METHOD metDI_RevisionSwitchOk
VAR_INPUT
    ITF_IN		:	CtaSysIO.ITF_IO;
END_VAR
VAR	
	ITF_DI		:	CtaSysIO.ITF_DI;
END_VAR
IF ITF_IN <> 0 THEN
	ITF_RevisionSwitchOk := ITF_IN;
	IF __QUERYINTERFACE(ITF_RevisionSwitchOk,ITF_DI) THEN
		xInActuatorRevisionSwitchOn := ITF_DI.proValue;
	END_IF
ELSE
	xInActuatorRevisionSwitchOn := 0;
END_IF
END_METHOD

PROPERTY proNotShowDI_RevisionSwitchOk : BOOL
GET
proNotShowDI_RevisionSwitchOk := NOT scParameter.scInSAtRevisionSwitch.fbxEnable.xValue OR scParameter.scInSAtRevisionSwitch.fbxInputMb.xValue;
END_GET
END_PROPERTY

PROPERTY proGetDI_RevisionSwitchOK : BOOL
GET
proGetDI_RevisionSwitchOK := xInActuatorRevisionSwitchOn;
END_GET
END_PROPERTY

PROPERTY proRevisionSwitch_ITF : CtaSysIO.ITF_IO
GET
proRevisionSwitch_ITF := ITF_RevisionSwitchOk;
END_GET
END_PROPERTY

PROPERTY proGetDI_FuseOK : BOOL
GET
proGetDI_FuseOK := xInFuseOk;
END_GET
END_PROPERTY

METHOD metDI_FuseOK
VAR_INPUT
    ITF_IN		:	CtaSysIO.ITF_IO;
END_VAR
VAR	
	ITF_DI		:	CtaSysIO.ITF_DI;
END_VAR
IF ITF_IN <> 0 THEN
	ITF_FuseOk := ITF_IN;
	IF __QUERYINTERFACE(ITF_FuseOk,ITF_DI) THEN
		xInFuseOk := ITF_DI.proValue;
	END_IF
ELSE
	xInFuseOk := 0;	
END_IF
END_METHOD

PROPERTY proNotShowDI_FuseOk : BOOL
GET
proNotShowDI_FuseOk := NOT scParameter.scFuse.fbxEnable.xValue OR scParameter.scFuse.fbxInputMb.xValue;
END_GET
END_PROPERTY

PROPERTY proFuse_ITF : CtaSysIO.ITF_IO
GET
proFuse_ITF := ITF_FuseOk;
END_GET
END_PROPERTY

METHOD metDI_ActuatorHand
VAR_INPUT
    ITF_IN		:	CtaSysIO.ITF_IO;
END_VAR
VAR	
	ITF_DI		:	CtaSysIO.ITF_DI;
END_VAR
IF ITF_IN <> 0 THEN
	ITF_ActuatorHand := ITF_IN;
	IF __QUERYINTERFACE(ITF_ActuatorHand,ITF_DI) THEN
		xInActuatorHand := ITF_DI.proValue;
	END_IF
ELSE	
	xInActuatorHand := 0;
END_IF
END_METHOD

PROPERTY proNotShowDI_ActuatorHand : BOOL
GET
proNotShowDI_ActuatorHand := NOT scParameter.scInSAtHand.fbxEnable.xValue OR scParameter.scInSAtHand.fbxInputMb.xValue;
END_GET
END_PROPERTY

PROPERTY proGetDI_ActuatorHand : BOOL
GET
proGetDI_ActuatorHand := xInActuatorHand;
END_GET
END_PROPERTY

PROPERTY proHandModul_ITF : CtaSysIO.ITF_IO
GET
proHandModul_ITF := ITF_ActuatorHand;
END_GET
END_PROPERTY

METHOD metDI_IsReady
VAR_INPUT
    ITF_IN		:	CtaSysIO.ITF_IO;
END_VAR
VAR	
	ITF_DI		:	CtaSysIO.ITF_DI;
END_VAR
IF ITF_IN <> 0 THEN
	ITF_ActuatorIsReady := ITF_IN;
	IF __QUERYINTERFACE(ITF_ActuatorIsReady,ITF_DI) THEN
		xInActuatorIsReady := ITF_DI.proValue;
	END_IF
ELSE
	xInActuatorIsReady := 0;
END_IF
END_METHOD

PROPERTY proNotShowDI_Ready : BOOL
GET
proNotShowDI_Ready := NOT scParameter.scInSAtReady.fbxEnable.xValue OR scParameter.scInSAtReady.fbxInputMb.xValue;
END_GET
END_PROPERTY

PROPERTY proGetDI_IsReady : BOOL
GET
proGetDI_IsReady := xInActuatorIsReady;
END_GET
END_PROPERTY

PROPERTY proActuatorReady_ITF : CtaSysIO.ITF_IO
GET
proActuatorReady_ITF := ITF_ActuatorIsReady;
END_GET
END_PROPERTY

PROPERTY proActuatorFuse_ITF : CtaSysIO.ITF_IO
GET
proActuatorFuse_ITF := ITF_ActuatorFuseOk;
END_GET
END_PROPERTY

METHOD metDI_ActuatorFuseOk
VAR_INPUT
    ITF_IN		:	CtaSysIO.ITF_IO;
END_VAR
VAR	
	ITF_DI		:	CtaSysIO.ITF_DI;
END_VAR
IF ITF_IN <> 0 THEN
	ITF_ActuatorFuseOk := ITF_IN;
	IF __QUERYINTERFACE(ITF_ActuatorFuseOk,ITF_DI) THEN
		xInActuatorFuseOk := ITF_DI.proValue;
	END_IF
ELSE	
	xInActuatorFuseOk := 0;
END_IF
END_METHOD

PROPERTY proNotShowDI_ActuatorFuseOk : BOOL
GET
proNotShowDI_ActuatorFuseOk := NOT scParameter.scActuatorFuse.fbxEnable.xValue OR scParameter.scActuatorFuse.fbxInputMb.xValue;
END_GET
END_PROPERTY

PROPERTY proGetDI_ActuatorFuseOk : BOOL
GET
proGetDI_ActuatorFuseOk := xInActuatorFuseOk;
END_GET
END_PROPERTY

METHOD metAI_ActualPosition
VAR_INPUT
    ITF_IN		:	CtaSysIO.ITF_IO;
END_VAR
VAR	
	ITF_AI		:	CtaSysIO.ITF_AI;
END_VAR
IF ITF_IN <> 0 THEN
	ITF_ActualPosition := ITF_IN;
	IF __QUERYINTERFACE(ITF_ActualPosition,ITF_AI) THEN
		rInActualPosition := ITF_AI.proValue;
	END_IF
ELSE	
	rInActualPosition := 0;
END_IF
END_METHOD

PROPERTY proNotShowAI_ActualPosition : BOOL
GET
proNotShowAI_ActualPosition := NOT scParameter.scInSAtActualPosition.fbxEnable.xValue OR scParameter.scInSAtActualPosition.fbxInputMb.xValue;
END_GET
END_PROPERTY

PROPERTY proGetAI_ActualPosition : REAL
GET
proGetAI_ActualPosition := rInActualPosition;
END_GET
END_PROPERTY

PROPERTY proActualPosition_ITF : CtaSysIO.ITF_IO
GET
proActualPosition_ITF := ITF_ActualPosition;
END_GET
END_PROPERTY

PROPERTY proOnY_ITF : CtaSysIO.ITF_IO
GET
proOnY_ITF := ITF_rOnY;
END_GET
END_PROPERTY

METHOD metAO_OnY : REAL
VAR_INPUT
    ITF_IN		:	CtaSysIO.ITF_IO;
END_VAR
VAR	
	ITF_AO		:	CtaSysIO.ITF_AO;
END_VAR
IF ITF_IN <> 0 THEN
	ITF_rOnY := ITF_IN;	
	IF __QUERYINTERFACE(ITF_rOnY,ITF_AO) THEN		
		ITF_AO.proValue := rOnY;
	END_IF	
ELSE
	metAO_OnY := rOnY;
END_IF
END_METHOD

METHOD metDO_xOnAuf : BOOL
VAR_INPUT
    ITF_IN		:	CtaSysIO.ITF_IO;
END_VAR
VAR	
	ITF_DO		:	CtaSysIO.ITF_DO;
END_VAR
IF ITF_IN <> 0 THEN	
	ITF_xOnAuf := ITF_IN;
	IF __QUERYINTERFACE(ITF_xOnAuf,ITF_DO) THEN		
		ITF_DO.proValue := xOnAuf;
	END_IF	
ELSE
	metDO_xOnAuf := xOnAuf;
END_IF
END_METHOD

PROPERTY proOnOpen_ITF : CtaSysIO.ITF_IO
GET
proOnOpen_ITF := ITF_xOnAuf;
END_GET
END_PROPERTY

PROPERTY proOnClose_ITF : CtaSysIO.ITF_IO
GET
proOnClose_ITF := ITF_xOnZu;
END_GET
END_PROPERTY

METHOD metDO_xOnZu : BOOL
VAR_INPUT
    ITF_IN		:	CtaSysIO.ITF_IO;
END_VAR
VAR	
	ITF_DO		:	CtaSysIO.ITF_DO;
END_VAR
IF ITF_IN <> 0 THEN	
	ITF_xOnZu := ITF_IN;
	IF __QUERYINTERFACE(ITF_xOnZu,ITF_DO) THEN		
		ITF_DO.proValue := xOnZu;
	END_IF	
ELSE
	metDO_xOnZu := xOnZu;
END_IF
END_METHOD

PROPERTY proOnY : REAL
GET
proOnY := rOnY;
END_GET
END_PROPERTY

ACTION actPrioOfControll:
(* get Controll request *)
xReleaseControllPrio := SEL(xRelease,xReleaseFromModBus,xRelease);  // xRelease request from Software has prio
rReleaseControllPrio := SEL(xRelease,rReleaseFromModBus,rRelease);  // rRelease request from Software has prio

(* Get state from Input or ModBus *)

(* Actuall Position from AI *)
// Value Actual Position 0 if not Enabled
rActualPosition						:= SEL(scParameter.scInSAtActualPosition.fbxEnable.xValue	,rOnY	,SEL(scParameter.scInSAtActualPosition.fbxInputMb.xValue	,rInActualPosition				,rInActualPositionMb			)); 
(* Actuator is Open *)
// Flag RückIsOpen False if not Enabled
xRückIsOpen							:= SEL(scParameter.scInSAtRükOpen.fbxEnable.xValue			,FALSE	,SEL(scParameter.scInSAtRükOpen.fbxInputMb.xValue			,xInRükIsOpen					,xInRükIsOpenMb					));
(* Actuator is Closed *)
// Flag RückIsClosed False if not Enabled
xRückIsClosed						:= SEL(scParameter.scInSAtRükClosed.fbxEnable.xValue		,FALSE	,SEL(scParameter.scInSAtRükClosed.fbxInputMb.xValue			,xInRükIsClosed					,xInRükIsClosedMb				));
(* Fuse ok *)
// Flag FuseOk True if not Enabled
xFuseOk								:= SEL(scParameter.scFuse.fbxEnable.xValue					,TRUE	,SEL(scParameter.scFuse.fbxInputMb.xValue					,xInFuseOk						,xInFuseOkMb                	));                     
(* Motor fuse ok *)
// Flag MotorFuseOk True if not Enabled
xActuatorFuseOk						:= SEL(scParameter.scActuatorFuse.fbxEnable.xValue			,TRUE	,SEL(scParameter.scActuatorFuse.fbxInputMb.xValue			,xInActuatorFuseOk				,xInActuatorFuseOkMb           	));
(* Motor is ready *)
// Flag MotorIsReady True if not Enabled
xActuatorIsReady					:= SEL(scParameter.scInSAtReady.fbxEnable.xValue			,TRUE	,SEL(scParameter.scInSAtReady.fbxInputMb.xValue				,xInActuatorIsReady				,xInActuatorIsReadyMb          	)); 
(* Revision Switch *)
// Flag MotorRevisionSwitchOn True if not Enabled
xActuatorRevisionSwitchOn			:= SEL(scParameter.scInSAtRevisionSwitch.fbxEnable.xValue	,TRUE	,SEL(scParameter.scInSAtRevisionSwitch.fbxInputMb.xValue	,xInActuatorRevisionSwitchOn	,xInActuatorRevisionSwitchOnMb 	));
xActuatorRevisionSwitchOff			:= NOT xActuatorRevisionSwitchOn;
(* Motor is hand *)
// Flag MotorHand False if not Enabled
xActuatorHand						:= SEL(scParameter.scInSAtHand.fbxEnable.xValue				,FALSE	,SEL(scParameter.scInSAtHand.fbxInputMb.xValue				,xInActuatorHand				,xInActuatorHandMb             	));
END_ACTION

ACTION actResetOnDisable:
TP_StartOeffnungVorlauf.PT  := T#0MS;
TP_StartOeffnungVorlauf.IN  := FALSE ;  
TP_StartOeffnungVorlauf();
                          
TP_Open.PT					:= T#0S;
TP_Open.IN					:= FALSE;
TP_Open();                  
TP_Close.PT					:= T#0S;  
TP_Close.IN					:= FALSE;
TP_Open();                  
                            
rActualPosition				:= 0	;
xRückIsOpen					:= FALSE;
xRückIsClosed				:= FALSE;
xFuseOk						:= FALSE;    
xActuatorFuseOk				:= FALSE;
xActuatorIsReady			:= FALSE;
xActuatorRevisionSwitchOn	:= FALSE;
xActuatorHand				:= FALSE;
END_ACTION

PROPERTY proOnAuf : BOOL
GET
proOnAuf := xOnAuf;
END_GET
END_PROPERTY

PROPERTY proOnZu : BOOL
GET
proOnZu := xOnZu;
END_GET
END_PROPERTY

//FB_Init ist immer implizit verfügbar und wird primär für die Initialisierung verwendet.
//Der Rückgabewert wird nicht ausgewertet. Für gezielte Einflussnahme können Sie
//die Methoden explizit deklarieren und darin mit dem Standard-Initialisierungscode 
//zusätzlichen Code bereitstellen. Sie können den Rückgabewert auswerten.
METHOD FB_INIT: BOOL
VAR_INPUT    
bInitRetains: BOOL; // TRUE: Die Retain-Variablen werden initialisiert (Reset warm / Reset kalt)    
bInCopyCode: BOOL;  // TRUE: Die Instanz wird danach in den Kopiercode kopiert (Online-Change)
END_VAR
VAR
    ITF_AT_THIS             :   ITF_STELLANTRIEB;
    ITF_AT_QUERRY           :   ITF_STELLANTRIEB;
END_VAR
IF NOT bInCopyCode THEN
    ITF_AT_THIS := THIS^;
    IF __QUERYINTERFACE(ITF_AT_THIS,ITF_AT_QUERRY) THEN
        diArrayPosition := GVL_StellAntrieb.fbStellAntrieb_Collector.metRegistry(ITF_AT_QUERRY);
    END_IF;
END_IF;
END_METHOD

PROPERTY proEn : BOOL
SET
xIsEnabled := proEn;
END_SET
GET
proEn := xIsEnabled;
END_GET
END_PROPERTY

PROPERTY proEnSymbol : STRING
GET
IF xIsEnabled THEN
    proEnSymbol := 'CtaVisSymbols.ImagePool.CheckboxChecked_blue';
ELSE    
    proEnSymbol := 'CtaVisSymbols.ImagePool.CheckboxUnchecked_withe'; 
END_IF;
END_GET
END_PROPERTY

ACTION actTrendLog:
(* Stellwert Digital zu *)		
fbTrendxOnZu.ENABLE 			:=	scParameter.scBase.fbxEnable.proValue AND
									scParameter.scInfluxDb.fbxEnable.proValue;
fbTrendxOnZu.KEY   				:= 	CONCAT(stObjID,'_xOnZu');
fbTrendxOnZu.SET_VALUE			:=	xOnZu;

(* Rückmeldung Digital zu *)
fbTrendxRückClosed.ENABLE 		:=	scParameter.scBase.fbxEnable.proValue AND
									scParameter.scInfluxDb.fbxEnable.proValue;
fbTrendxRückClosed.KEY   		:= 	CONCAT(stObjID,'_xRückIsClosed');
fbTrendxRückClosed.SET_VALUE	:=	xRückIsClosed;

(* Stellwert Digital auf *)
fbTrendxOnAuf.ENABLE 			:=	scParameter.scBase.fbxEnable.proValue AND
									scParameter.scInfluxDb.fbxEnable.proValue;
fbTrendxOnAuf.KEY   			:= 	CONCAT(stObjID,'_xOnAuf');
fbTrendxOnAuf.SET_VALUE			:=	xOnAuf;

(* Rückmeldung Digital auf *)
fbTrendxRückIsOpen.ENABLE 		:=	scParameter.scBase.fbxEnable.proValue AND
									scParameter.scInfluxDb.fbxEnable.proValue;
fbTrendxRückIsOpen.KEY   		:= 	CONCAT(stObjID,'_xRückIsOpen');
fbTrendxRückIsOpen.SET_VALUE	:=	xRückIsOpen;

(* Stellwert Analog *)
fbTrendrOnY.ENABLE 				:=	scParameter.scBase.fbxEnable.proValue AND
									scParameter.scInfluxDb.fbxEnable.proValue;
fbTrendrOnY.KEY   				:= 	CONCAT(stObjID,'_rOnY');
fbTrendrOnY.SET_VALUE			:=	rOnY;

(* Istwert Analog *)
fbTrendrIsOnY.ENABLE 			:=	scParameter.scBase.fbxEnable.proValue AND
									scParameter.scInfluxDb.fbxEnable.proValue;
fbTrendrIsOnY.KEY   			:= 	CONCAT(stObjID,'_rIsOnY');
fbTrendrIsOnY.SET_VALUE			:=	proIsOnY;

(* Fehler *)
fbTrendxError.ENABLE 			:=	scParameter.scBase.fbxEnable.proValue AND
									scParameter.scInfluxDb.fbxEnable.proValue;
fbTrendxError.KEY   			:= 	CONCAT(stObjID,'_xError');
fbTrendxError.SET_VALUE			:=	xIsError;
END_ACTION

ACTION actReport:
(* EWI Manager *)
fbReportManager(	stErrorInitReportTextListIn		:=	ADR(GlobalKonstant.stReportTextListError),
					stWarningInitReportTextListIn	:=	ADR(GlobalKonstant.stReportTextListWarning),
					stInfoInitReportTextListIn		:=	ADR(GlobalKonstant.stReportTextListInfo),
					scReportNr						:=	scEWI);
(* Errors *)                        
		(* Stellwert Rückmeldung *)
		ayErrorReporter[1].proPrio  := 3;
		ayErrorReporter[1].metReport(     		xSetReportIn					:= xErrorDiffAI AND scParameter.scInSAtActualPosition.fbxDoesAlarm.proValue AND scParameter.scInSAtActualPosition.fbxEnable.proValue,
												iReportID						:= 1,
												enReportTypeIn					:= CtaAppReport.enReportType.Error,  
												enReportAcknowledgeTypeIn   	:= scParameter.scInSAtActualPosition.fbiTypeOfAck.proValue,
												tDelay							:= T#0S, 
												ITF_BMK_IN						:= THIS^,			              
												pstReportTextListIn				:= ADR(GlobalKonstant.stReportTextListError),
												stOptionalReportText		    := '',   
												iRetryTilReportLock 		    := scParameter.scInSAtActualPosition.fbiMaxErrorRetryAllowed.proValue, 
												xResetCount         		    := FALSE,  
												tReset						    := T#24H); 		

		(* Stellventil keine rückmeldung Zu *) 
		ayErrorReporter[2].proPrio  := 3;   
        ayErrorReporter[2].metReport(     		xSetReportIn					:= xErrorCloseDI AND scParameter.scInSAtRükClosed.fbxDoesAlarm.proValue AND scParameter.scInSAtRükClosed.fbxEnable.proValue,
												iReportID						:= 2,
												enReportTypeIn					:= CtaAppReport.enReportType.Error,  
												enReportAcknowledgeTypeIn   	:= scParameter.scInSAtRükClosed.fbiTypeOfAck.proValue,
												tDelay							:= T#0S, 
												ITF_BMK_IN						:= THIS^,			              
												pstReportTextListIn				:= ADR(GlobalKonstant.stReportTextListError),
												stOptionalReportText		    := '',   
												iRetryTilReportLock 		    := scParameter.scInSAtRükClosed.fbiMaxErrorRetryAllowed.proValue, 
												xResetCount         		    := FALSE,  
												tReset						    := T#24H); 	  
		(* Stellventil keine rückmeldung Auf *)
		ayErrorReporter[3].proPrio  := 3; 
		ayErrorReporter[3].metReport(     		xSetReportIn					:= xErrorOpenDI AND scParameter.scInSAtRükOpen.fbxDoesAlarm.proValue AND scParameter.scInSAtRükOpen.fbxEnable.proValue,
												iReportID						:= 3,
												enReportTypeIn					:= CtaAppReport.enReportType.Error,  
												enReportAcknowledgeTypeIn   	:= scParameter.scInSAtRükOpen.fbiTypeOfAck.proValue,
												tDelay							:= T#1S, 
												ITF_BMK_IN						:= THIS^,			              
												pstReportTextListIn				:= ADR(GlobalKonstant.stReportTextListError),
												stOptionalReportText		    := '',   
												iRetryTilReportLock 		    := scParameter.scInSAtRükOpen.fbiMaxErrorRetryAllowed.proValue, 
												xResetCount         		    := FALSE,  
												tReset						    := T#24H);
		(* Monitoring digitaler Stellwert *)
		ayErrorReporter[4].proPrio  := 3;    
		ayErrorReporter[4].metReport(     		xSetReportIn					:= xErrorDiRük AND scParameter.scBase.fbxEnDigitalMonitoring.proValue,
												iReportID						:= 4,
												enReportTypeIn					:= CtaAppReport.enReportType.Error,  
												enReportAcknowledgeTypeIn   	:= CtaAppReport.enReportacknowledgeType.Auto,
												tDelay							:= T#1S, 
												ITF_BMK_IN						:= THIS^,			              
												pstReportTextListIn				:= ADR(GlobalKonstant.stReportTextListError),
												stOptionalReportText		    := '',   
												iRetryTilReportLock 		    := 0, 
												xResetCount         		    := FALSE,  
												tReset						    := T#24H);
		(* Monitoring analoger Stellwert *)
		ayErrorReporter[5].proPrio  := 3;     
		ayErrorReporter[5].metReport(     		xSetReportIn					:= xErrorAIRük AND scParameter.scBase.fbxEnAnalogMonitoring.proValue,
												iReportID						:= 5,
												enReportTypeIn					:= CtaAppReport.enReportType.Error,  
												enReportAcknowledgeTypeIn   	:= CtaAppReport.enReportacknowledgeType.Auto,
												tDelay							:= T#1S, 
												ITF_BMK_IN						:= THIS^,			              
												pstReportTextListIn				:= ADR(GlobalKonstant.stReportTextListError),
												stOptionalReportText		    := '',   
												iRetryTilReportLock 		    := 0, 
												xResetCount         		    := FALSE,  
												tReset						    := T#24H);                    
		(* Error Fuse *)
		ayErrorReporter[6].proPrio  := 2;    
		ayErrorReporter[6].metReport(     		xSetReportIn					:= NOT xFuseOk AND scParameter.scFuse.fbxDoesAlarm.proValue AND scParameter.scFuse.fbxEnable.proValue,
												iReportID						:= 6,
												enReportTypeIn					:= CtaAppReport.enReportType.Error,  
												enReportAcknowledgeTypeIn   	:= CtaAppReport.enReportacknowledgeType.Auto,
												tDelay							:= T#1S, 
												ITF_BMK_IN						:= THIS^,			              
												pstReportTextListIn				:= ADR(GlobalKonstant.stReportTextListError),
												stOptionalReportText		    := '',   
												iRetryTilReportLock 		    := 0, 
												xResetCount         		    := FALSE,  
												tReset						    := T#24H);
                                                
		(* Error Actuator Fuse *)
		ayErrorReporter[7].proPrio  := 2;    
		ayErrorReporter[7].metReport(     		xSetReportIn					:= NOT xActuatorFuseOk AND scParameter.scActuatorFuse.fbxDoesAlarm.proValue AND scParameter.scActuatorFuse.fbxEnable.proValue,
												iReportID						:= 7,
												enReportTypeIn					:= CtaAppReport.enReportType.Error,  
												enReportAcknowledgeTypeIn   	:= CtaAppReport.enReportacknowledgeType.Auto,
												tDelay							:= T#1S, 
												ITF_BMK_IN						:= THIS^,			              
												pstReportTextListIn				:= ADR(GlobalKonstant.stReportTextListError),
												stOptionalReportText		    := '',   
												iRetryTilReportLock 		    := 0, 
												xResetCount         		    := FALSE,  
												tReset						    := T#24H);                                                

		(* Config Error *)
		ayErrorReporter[8].proPrio  := 1;    
		ayErrorReporter[8].metReport(     		xSetReportIn					:= xConfigError,
												iReportID						:= 8,
												enReportTypeIn					:= CtaAppReport.enReportType.Error,  
												enReportAcknowledgeTypeIn   	:= CtaAppReport.enReportacknowledgeType.Quit,
												tDelay							:= T#1S, 
												ITF_BMK_IN						:= THIS^,			              
												pstReportTextListIn				:= ADR(GlobalKonstant.stReportTextListError),
												stOptionalReportText		    := '',   
												iRetryTilReportLock 		    := 0, 
												xResetCount         		    := FALSE,  
												tReset						    := T#24H);                                           
(* Warnungen *)
		(* Warnung Revisionsschalter Aus *)
		ayWarningReporter[1].proPrio  := 1;
		ayWarningReporter[1].proHandLokal :=   	xActuatorRevisionSwitchOff; 
		ayWarningReporter[1].metReport(			xSetReportIn					:= xActuatorRevisionSwitchOff,
												iReportID						:= 1,
												enReportTypeIn					:= CtaAppReport.enReportType.Warning,  
												enReportAcknowledgeTypeIn   	:= CtaAppReport.enReportAcknowledgeType.Auto,
												tDelay							:= T#0S, 
												ITF_BMK_IN						:= THIS^,			              
												pstReportTextListIn				:= ADR(GlobalKonstant.stReportTextListWarning),
												stOptionalReportText		    := '',   
												iRetryTilReportLock 		    := 0, 
												xResetCount         		    := FALSE,  
												tReset						    := T#0S);     

		(* Warnung Hand Aus *)
		ayWarningReporter[2].proPrio  := 3;        
		ayWarningReporter[2].proHandLokal :=    xIsHandOff; 
		ayWarningReporter[2].metReport(			xSetReportIn					:= xIsHandOff,
												iReportID						:= 2,
												enReportTypeIn					:= CtaAppReport.enReportType.Warning,  
												enReportAcknowledgeTypeIn   	:= CtaAppReport.enReportAcknowledgeType.Auto,
												tDelay							:= T#0S, 
												ITF_BMK_IN						:= THIS^,			              
												pstReportTextListIn				:= ADR(GlobalKonstant.stReportTextListWarning),
												stOptionalReportText		    := '',   
												iRetryTilReportLock 		    := 0, 
												xResetCount         		    := FALSE,  
												tReset						    := T#0S);                                  
                                
        (* Warnung Hand Ein *)
		ayWarningReporter[3].proPrio  := 3;    
		ayWarningReporter[3].proHandLokal :=    xIsHandOn;
		ayWarningReporter[3].metReport(			xSetReportIn					:= xIsHandOn,
												iReportID						:= 3,
												enReportTypeIn					:= CtaAppReport.enReportType.Warning,  
												enReportAcknowledgeTypeIn   	:= CtaAppReport.enReportAcknowledgeType.Auto,
												tDelay							:= T#0S, 
												ITF_BMK_IN						:= THIS^,			              
												pstReportTextListIn				:= ADR(GlobalKonstant.stReportTextListWarning),
												stOptionalReportText		    := '',   
												iRetryTilReportLock 		    := 0, 
												xResetCount         		    := FALSE,  
												tReset						    := T#0S);   
 
        (* Warnung Handmodul Actuator *)
		ayWarningReporter[4].proPrio  := 4;    
		ayWarningReporter[4].proHandLokal :=    xActuatorHand;
		ayWarningReporter[4].metReport(			xSetReportIn					:= xActuatorHand,
												iReportID						:= 4,
												enReportTypeIn					:= CtaAppReport.enReportType.Warning,  
												enReportAcknowledgeTypeIn   	:= CtaAppReport.enReportAcknowledgeType.Auto,
												tDelay							:= T#0S, 
												ITF_BMK_IN						:= THIS^,			              
												pstReportTextListIn				:= ADR(GlobalKonstant.stReportTextListWarning),
												stOptionalReportText		    := '',   
												iRetryTilReportLock 		    := 0, 
												xResetCount         		    := FALSE,  
												tReset						    := T#0S);                                                   
(* Sync Reports *)                                         
FOR difor := LOWER_BOUND(ayErrorReporter,1) TO UPPER_BOUND(ayErrorReporter,1) DO
	fbReportManager.metSyncReporter(ayErrorReporter[difor]);	
END_FOR;
FOR difor := LOWER_BOUND(ayWarningReporter,1) TO UPPER_BOUND(ayWarningReporter,1) DO
	fbReportManager.metSyncReporter(ayWarningReporter[difor]);	
END_FOR;
                                                                             
_xIsError   := scEWI.iError <> 0;
_xIsWarning := scEWI.iWarning <> 0;
END_ACTION

{attribute 'monitoring' := 'variable'}
PROPERTY proAcknowlege : BOOL
GET
proAcknowlege := NOT proIsError;
END_GET
END_PROPERTY

{attribute 'monitoring' := 'variable'}
PROPERTY proAvailable : BOOL
GET
proAvailable := proIsReady;
END_GET
END_PROPERTY

{attribute 'monitoring' := 'variable'}
PROPERTY proLockDown : BOOL
GET
proLockDown := proIsError;
END_GET
END_PROPERTY

END_FUNCTION_BLOCK

// 30 Program Organization Units/Abstracte Bausteine/fbAntriebTabellenInfo
{attribute 'hide'} 
FUNCTION_BLOCK INTERNAL ABSTRACT fbAntriebTabellenInfo EXTENDS CtaAppBmk.fbBMK IMPLEMENTS ITF_STELLANTRIEB_TABELLE_INFO

PROPERTY proOnAuf : BOOL
GET
END_GET
END_PROPERTY

PROPERTY proStateSymbol : STRING
GET
END_GET
END_PROPERTY

PROPERTY proEnSymbol : STRING
GET
END_GET
END_PROPERTY

PROPERTY proIsOn : BOOL
GET
END_GET
END_PROPERTY

PROPERTY proIsOnY : REAL
GET
END_GET
END_PROPERTY

PROPERTY proOn : BOOL
GET
END_GET
END_PROPERTY

PROPERTY proOnY : REAL
GET
END_GET
END_PROPERTY

PROPERTY proOnZu : BOOL
GET
END_GET
END_PROPERTY

PROPERTY proRükIsClosed : BOOL
GET
END_GET
END_PROPERTY

PROPERTY proRükIsOpen : BOOL
GET
END_GET
END_PROPERTY

END_FUNCTION_BLOCK

// 21 Interface/ITF_STELLANTRIEB_TABELLE_INFO
INTERFACE INTERNAL ITF_STELLANTRIEB_TABELLE_INFO EXTENDS CtaAppBmk.ITF_BMK

PROPERTY proRükIsOpen : BOOL
GET
END_GET
END_PROPERTY

PROPERTY proRükIsClosed : BOOL
GET
END_GET
END_PROPERTY

PROPERTY INTERNAL proStateSymbol : STRING
GET
END_GET
END_PROPERTY

PROPERTY INTERNAL proEnSymbol : STRING
GET
END_GET
END_PROPERTY

PROPERTY proOnZu : BOOL
GET
END_GET
END_PROPERTY

PROPERTY proIsOnY : REAL
GET
END_GET
END_PROPERTY

PROPERTY proOnAuf : BOOL
GET
END_GET
END_PROPERTY

PROPERTY proOnY : REAL
GET
END_GET
END_PROPERTY

END_INTERFACE

// 21 Interface/ITF_STELLANTRIEB
INTERFACE ITF_STELLANTRIEB EXTENDS ITF_STELLANTRIEB_TABELLE_INFO,CtaAppModbusSpezifikation.ITF_MODBUS_SPEZIFIKATION

PROPERTY proAuto : BOOL
GET
END_GET
SET
END_SET
END_PROPERTY

PROPERTY proHandOff : BOOL
GET
END_GET
SET
END_SET
END_PROPERTY

PROPERTY proHandOn : BOOL
GET
END_GET
SET
END_SET
END_PROPERTY

PROPERTY proIsRegulatet : BOOL
GET
END_GET
END_PROPERTY

PROPERTY proIsError : BOOL
GET
END_GET
END_PROPERTY

PROPERTY proIsWarning : BOOL
GET
END_GET
END_PROPERTY

PROPERTY proIsEnabled : BOOL
GET
END_GET
END_PROPERTY

PROPERTY proIsHandOnOrOff : BOOL
GET
END_GET
END_PROPERTY

PROPERTY proIsReady : BOOL
GET
END_GET
END_PROPERTY

PROPERTY proHardWareHandModulAktive : BOOL
GET
END_GET
END_PROPERTY

PROPERTY proRevisionSwitchOk : BOOL
GET
END_GET
END_PROPERTY

PROPERTY proHandOnY : REAL
SET
END_SET
GET
END_GET
END_PROPERTY

PROPERTY proEn : BOOL
SET
END_SET
GET
END_GET
END_PROPERTY

PROPERTY proGetDI_RükIsOpen : BOOL
GET
END_GET
END_PROPERTY

PROPERTY proNotShowDI_RükIsOpen : BOOL
GET
END_GET
END_PROPERTY

PROPERTY proIsOpen_ITF : CtaSysIO.ITF_IO
GET
END_GET
END_PROPERTY

PROPERTY INTERNAL proGetDI_ActuatorHand : BOOL
GET
END_GET
END_PROPERTY

PROPERTY proNotShowDI_ActuatorHand : BOOL
GET
END_GET
END_PROPERTY

PROPERTY proHandModul_ITF : CtaSysIO.ITF_IO
GET
END_GET
END_PROPERTY

PROPERTY INTERNAL proGetDI_ActuatorFuseOk : BOOL
GET
END_GET
END_PROPERTY

PROPERTY proNotShowDI_ActuatorFuseOk : BOOL
GET
END_GET
END_PROPERTY

PROPERTY proActuatorFuse_ITF : CtaSysIO.ITF_IO
GET
END_GET
END_PROPERTY

PROPERTY INTERNAL proGetDI_IsReady : BOOL
GET
END_GET
END_PROPERTY

PROPERTY proNotShowDI_Ready : BOOL
GET
END_GET
END_PROPERTY

PROPERTY proActuatorReady_ITF : CtaSysIO.ITF_IO
GET
END_GET
END_PROPERTY

PROPERTY INTERNAL proGetDI_FuseOK : BOOL
GET
END_GET
END_PROPERTY

PROPERTY proNotShowDI_FuseOk : BOOL
GET
END_GET
END_PROPERTY

PROPERTY proFuse_ITF : CtaSysIO.ITF_IO
GET
END_GET
END_PROPERTY

PROPERTY INTERNAL proGetDI_RevisionSwitchOK : BOOL
GET
END_GET
END_PROPERTY

PROPERTY proNotShowDI_RevisionSwitchOk : BOOL
GET
END_GET
END_PROPERTY

PROPERTY proRevisionSwitch_ITF : CtaSysIO.ITF_IO
GET
END_GET
END_PROPERTY

PROPERTY proNotShowAI_ActualPosition : BOOL
GET
END_GET
END_PROPERTY

PROPERTY proGetAI_ActualPosition : REAL
GET
END_GET
END_PROPERTY

PROPERTY proActualPosition_ITF : CtaSysIO.ITF_IO
GET
END_GET
END_PROPERTY

PROPERTY proGetDI_RükIsClosed : BOOL
GET
END_GET
END_PROPERTY

PROPERTY proNotShowDI_RükIsClosed : BOOL
GET
END_GET
END_PROPERTY

PROPERTY proIsClosed_ITF : CtaSysIO.ITF_IO
GET
END_GET
END_PROPERTY

PROPERTY proOnOpen_ITF : CtaSysIO.ITF_IO
GET
END_GET
END_PROPERTY

PROPERTY proOnClose_ITF : CtaSysIO.ITF_IO
GET
END_GET
END_PROPERTY

PROPERTY proOnY_ITF : CtaSysIO.ITF_IO
GET
END_GET
END_PROPERTY

PROPERTY INTERNAL proAnzWarning : INT
GET
END_GET
END_PROPERTY

PROPERTY INTERNAL proITF_REPORTMANAGER : CtaAppReport.ITF_REPORTMANAGER
GET
END_GET
END_PROPERTY

PROPERTY INTERNAL proAnzInfo : INT
GET
END_GET
END_PROPERTY

PROPERTY INTERNAL proAnzError : INT
GET
END_GET
END_PROPERTY

PROPERTY INTERNAL proModbusTest : BOOL
SET
END_SET
GET
END_GET
END_PROPERTY

PROPERTY proModbusStateWord : REFERENCE TO ARRAY[0..3] OF WORD
GET
END_GET
END_PROPERTY

PROPERTY proModbusControllWord : REFERENCE TO ARRAY[0..3] OF WORD
GET
END_GET
END_PROPERTY

PROPERTY proConfigError : BOOL
GET
END_GET
END_PROPERTY

PROPERTY p_scActuatorFuse_fbxEnable : CtaSysConfig.ITF_DATATYPE;
GET
END_GET
END_PROPERTY

PROPERTY p_scActuatorFuse_fbxInputMb : CtaSysConfig.ITF_DATATYPE;
GET
END_GET
END_PROPERTY

PROPERTY p_scActuatorFuse_fbxDoesAlarm : CtaSysConfig.ITF_DATATYPE;
GET
END_GET
END_PROPERTY

PROPERTY p_scBase_fbxEnable : CtaSysConfig.ITF_DATATYPE;
GET
END_GET
END_PROPERTY

PROPERTY p_scBase_fbxControllMb : CtaSysConfig.ITF_DATATYPE;
GET
END_GET
END_PROPERTY

PROPERTY p_scBase_fbxInvertiert : CtaSysConfig.ITF_DATATYPE;
GET
END_GET
END_PROPERTY

PROPERTY p_scBase_fbxRegulatet : CtaSysConfig.ITF_DATATYPE;
GET
END_GET
END_PROPERTY

PROPERTY p_scBase_fbrYMin : CtaSysConfig.ITF_DATATYPE;
GET
END_GET
END_PROPERTY

PROPERTY p_scBase_fbrYMax : CtaSysConfig.ITF_DATATYPE;
GET
END_GET
END_PROPERTY

PROPERTY p_scBase_fbxEnStartPosition : CtaSysConfig.ITF_DATATYPE;
GET
END_GET
END_PROPERTY

PROPERTY p_scBase_fbrYStartPos : CtaSysConfig.ITF_DATATYPE;
GET
END_GET
END_PROPERTY

PROPERTY p_scBase_fbtStartPosTime : CtaSysConfig.ITF_DATATYPE;
GET
END_GET
END_PROPERTY

PROPERTY p_scBase_fbrYStopp : CtaSysConfig.ITF_DATATYPE;
GET
END_GET
END_PROPERTY

PROPERTY p_scBase_fbtYSettingTime : CtaSysConfig.ITF_DATATYPE;
GET
END_GET
END_PROPERTY

PROPERTY p_scBase_fbxEnDigitalValve : CtaSysConfig.ITF_DATATYPE;
GET
END_GET
END_PROPERTY

PROPERTY p_scBase_fbrHysteresisDigital : CtaSysConfig.ITF_DATATYPE;
GET
END_GET
END_PROPERTY

PROPERTY p_scBase_fbrRefIsOpen : CtaSysConfig.ITF_DATATYPE;
GET
END_GET
END_PROPERTY

PROPERTY p_scBase_fbrRefIsClosed : CtaSysConfig.ITF_DATATYPE;
GET
END_GET
END_PROPERTY

PROPERTY p_scBase_fbxEnDigitalMonitoring : CtaSysConfig.ITF_DATATYPE;
GET
END_GET
END_PROPERTY

PROPERTY p_scBase_fbxEnAnalogMonitoring : CtaSysConfig.ITF_DATATYPE;
GET
END_GET
END_PROPERTY

PROPERTY p_scFuse_fbxEnable : CtaSysConfig.ITF_DATATYPE;
GET
END_GET
END_PROPERTY

PROPERTY p_scFuse_fbxInputMb : CtaSysConfig.ITF_DATATYPE;
GET
END_GET
END_PROPERTY

PROPERTY p_scFuse_fbxDoesAlarm : CtaSysConfig.ITF_DATATYPE;
GET
END_GET
END_PROPERTY

PROPERTY p_scInStellAtRevisionSwitch_fbxEnable : CtaSysConfig.ITF_DATATYPE;
GET
END_GET
END_PROPERTY

PROPERTY p_scInStellAtRevisionSwitch_fbxInputMb : CtaSysConfig.ITF_DATATYPE;
GET
END_GET
END_PROPERTY

PROPERTY p_scInStellAtReady_fbxEnable : CtaSysConfig.ITF_DATATYPE;
GET
END_GET
END_PROPERTY

PROPERTY p_scInStellAtReady_fbxInputMb : CtaSysConfig.ITF_DATATYPE;
GET
END_GET
END_PROPERTY

PROPERTY p_scInStellAtHand_fbxEnable : CtaSysConfig.ITF_DATATYPE;
GET
END_GET
END_PROPERTY

PROPERTY p_scInStellAtHand_fbxInputMb : CtaSysConfig.ITF_DATATYPE;
GET
END_GET
END_PROPERTY

PROPERTY p_scInStellAtRükClosed_fbxEnable : CtaSysConfig.ITF_DATATYPE;
GET
END_GET
END_PROPERTY

PROPERTY p_scInStellAtRükClosed_fbxInputMb : CtaSysConfig.ITF_DATATYPE;
GET
END_GET
END_PROPERTY

PROPERTY p_scInStellAtRükClosed_fbxDoesAlarm : CtaSysConfig.ITF_DATATYPE;
GET
END_GET
END_PROPERTY

PROPERTY p_scInStellAtRükClosed_fbtDelayStart : CtaSysConfig.ITF_DATATYPE;
GET
END_GET
END_PROPERTY

PROPERTY p_scInStellAtRükClosed_fbtDelayRun : CtaSysConfig.ITF_DATATYPE;
GET
END_GET
END_PROPERTY

PROPERTY p_scInStellAtRükClosed_fbiTypeOfAck : CtaSysConfig.ITF_DATATYPE;
GET
END_GET
END_PROPERTY

PROPERTY p_scInStellAtRükClosed_fbiMaxErrorRetryAllowed : CtaSysConfig.ITF_DATATYPE;
GET
END_GET
END_PROPERTY

PROPERTY p_scInStellAtRükOpen_fbxEnable : CtaSysConfig.ITF_DATATYPE;
GET
END_GET
END_PROPERTY

PROPERTY p_scInStellAtRükOpen_fbxInputMb : CtaSysConfig.ITF_DATATYPE;
GET
END_GET
END_PROPERTY

PROPERTY p_scInStellAtRükOpen_fbxDoesAlarm : CtaSysConfig.ITF_DATATYPE;
GET
END_GET
END_PROPERTY

PROPERTY p_scInStellAtRükOpen_fbtDelayStart : CtaSysConfig.ITF_DATATYPE;
GET
END_GET
END_PROPERTY

PROPERTY p_scInStellAtRükOpen_fbtDelayRun : CtaSysConfig.ITF_DATATYPE;
GET
END_GET
END_PROPERTY

PROPERTY p_scInStellAtRükOpen_fbiTypeOfAck : CtaSysConfig.ITF_DATATYPE;
GET
END_GET
END_PROPERTY

PROPERTY p_scInStellAtRükOpen_fbiMaxErrorRetryAllowed : CtaSysConfig.ITF_DATATYPE;
GET
END_GET
END_PROPERTY

PROPERTY p_scInStellAtActualPosition_fbxEnable : CtaSysConfig.ITF_DATATYPE;
GET
END_GET
END_PROPERTY

PROPERTY p_scInStellAtActualPosition_fbxInputMb : CtaSysConfig.ITF_DATATYPE;
GET
END_GET
END_PROPERTY

PROPERTY p_scInStellAtActualPosition_fbxDoesAlarm : CtaSysConfig.ITF_DATATYPE;
GET
END_GET
END_PROPERTY

PROPERTY p_scInStellAtActualPosition_fbrMaxDiff : CtaSysConfig.ITF_DATATYPE;
GET
END_GET
END_PROPERTY

PROPERTY p_scInStellAtActualPosition_fbtDelayStart : CtaSysConfig.ITF_DATATYPE;
GET
END_GET
END_PROPERTY

PROPERTY p_scInStellAtActualPosition_fbtDelayRun : CtaSysConfig.ITF_DATATYPE;
GET
END_GET
END_PROPERTY

PROPERTY p_scInStellAtActualPosition_fbiTypeOfAck : CtaSysConfig.ITF_DATATYPE;
GET
END_GET
END_PROPERTY

PROPERTY p_scInStellAtActualPosition_fbiMaxErrorRetryAllowed : CtaSysConfig.ITF_DATATYPE;
GET
END_GET
END_PROPERTY

PROPERTY p_scManual_fbxAlowManualOn : CtaSysConfig.ITF_DATATYPE;
GET
END_GET
END_PROPERTY

PROPERTY p_scManual_fbuiManualState : CtaSysConfig.ITF_DATATYPE;
GET
END_GET
END_PROPERTY

PROPERTY p_scManual_fbrManualOnY : CtaSysConfig.ITF_DATATYPE;
GET
END_GET
END_PROPERTY

PROPERTY p_scInfluxDb_fbxEnable : CtaSysConfig.ITF_DATATYPE;
GET
END_GET
END_PROPERTY

PROPERTY proRefToRonYDumper : REFERENCE TO CtaAppDumper.fbDumper
GET
END_GET
END_PROPERTY

PROPERTY proIsInverted : BOOL
GET
END_GET
END_PROPERTY

PROPERTY proValveIcon : UINT
GET
END_GET
SET
END_SET
END_PROPERTY

{attribute 'monitoring' := 'variable'}
PROPERTY proAcknowlege : BOOL
GET
END_GET
END_PROPERTY

{attribute 'monitoring' := 'variable'}
PROPERTY proAvailable : BOOL
GET
END_GET
END_PROPERTY

{attribute 'monitoring' := 'variable'}
PROPERTY proLockDown : BOOL
GET
END_GET
END_PROPERTY

PROPERTY proOn : BOOL
GET
END_GET
END_PROPERTY

END_INTERFACE

// 30 Program Organization Units/fbStellAntrieb_Collector
FUNCTION_BLOCK fbStellAntrieb_Collector IMPLEMENTS ITF_STELLANTRIEB_COLLECTOR
VAR_INPUT
END_VAR
VAR_OUTPUT
END_VAR
VAR
    ayAT_INTERFACE          : ARRAY[1..Parameter.iMaxStellAntrieb] OF ITF_STELLANTRIEB;   
    ayAT_INTERFACE_SORTET   : ARRAY[1..Parameter.iMaxStellAntrieb] OF ITF_STELLANTRIEB; 
    xIsSortet               : BOOL;
    diNext                  : DINT    := 1;
    diMin                   : DINT    := 1;
    diMax                   : DINT;
    diMaxSort               : DINT;
    xError                  : BOOL;
    xBufferError            : BOOL;
    diMissedBuffer          : DINT;
END_VAR

METHOD metRegistry : DINT
VAR_INPUT
    ITF_AT_IN   :   ITF_STELLANTRIEB;
END_VAR
VAR
    diArrayPos  :   DINT;
    diCount     :   DINT;
END_VAR
IF ITF_AT_IN <> 0 THEN
    diArrayPos := __XADD(ADR(diNext),1);
    IF diArrayPos <= Parameter.iMaxStellAntrieb AND diArrayPos >= 1 THEN
        IF __QUERYINTERFACE(ITF_AT_IN,ayAT_INTERFACE[diArrayPos]) THEN
            metRegistry             := diArrayPos;
            GVL_StellAntrieb.xValidData       := TRUE;
            diCount    := __XADD(ADR(diMax),1);
        END_IF;
    ELSE
        IF diArrayPos > Parameter.iMaxStellAntrieb THEN
            xBufferError := TRUE;
            diMissedBuffer := diArrayPos - Parameter.iMaxStellAntrieb;
		END_IF;
        xError      := TRUE; 
        metRegistry := 0;
    END_IF;   
ELSE
    xError := TRUE; 
    metRegistry := 0;
END_IF;
END_METHOD

METHOD metSortArray
VAR_INPUT
    stSearch    :   STRING;
    uiSort      :   UINT;
END_VAR
VAR
    diFor1      :   DINT;
    diFor2      :   DINT;
    diFill      :   DINT;
    ITF_AT_Temp :   ITF_STELLANTRIEB;    
    iBigger     :   INT;
END_VAR
IF stSearch <> '' THEN
    diMaxSort   := 0;
    diFill      := LOWER_BOUND(ayAT_INTERFACE,1); 
    FOR diFor1 := LOWER_BOUND(ayAT_INTERFACE,1) TO UPPER_BOUND(ayAT_INTERFACE,1) DO
        IF ayAT_INTERFACE[diFor1] <> 0 THEN
            IF FIND(ayAT_INTERFACE[diFor1].proGetBMK,stSearch) <> 0 OR FIND(ayAT_INTERFACE[diFor1].proGetVendorDesignation,stSearch) <> 0 THEN
                ayAT_INTERFACE_SORTET[diFill] := ayAT_INTERFACE[diFor1];
                diFill      := diFill + 1; 
                diMaxSort   := diFill -1; 
            END_IF;
        END_IF;
	END_FOR;
ELSE
    ayAT_INTERFACE_SORTET := ayAT_INTERFACE;
    diMaxSort := diMax;
END_IF; 
// 1 = Sort BMK
IF uiSort = 1 THEN
    FOR diFor1 := LOWER_BOUND(ayAT_INTERFACE_SORTET,1) TO diMaxSort DO 
        FOR diFor2 := LOWER_BOUND(ayAT_INTERFACE_SORTET,1) TO diMaxSort -1 DO 
            IF ayAT_INTERFACE_SORTET[diFor2] <> 0 AND ayAT_INTERFACE_SORTET[diFor2 + 1] <> 0 THEN
                IF LEN(ayAT_INTERFACE_SORTET[diFor2].proGetBMK) > LEN(ayAT_INTERFACE_SORTET[diFor2 + 1].proGetBMK) THEN
                    ITF_AT_Temp                         := ayAT_INTERFACE_SORTET[diFor2];
                    ayAT_INTERFACE_SORTET[diFor2]       := ayAT_INTERFACE_SORTET[diFor2 + 1];
                    ayAT_INTERFACE_SORTET[diFor2 + 1]   := ITF_AT_Temp; 
                ELSIF LEN(ayAT_INTERFACE_SORTET[diFor2].proGetBMK) = LEN(ayAT_INTERFACE_SORTET[diFor2 + 1].proGetBMK) THEN
                    iBigger := fcGetBigerStringValue(ayAT_INTERFACE_SORTET[diFor2].proGetBMK,ayAT_INTERFACE_SORTET[diFor2 + 1].proGetBMK);
                    IF iBigger = 1 THEN
                        ITF_AT_Temp                         := ayAT_INTERFACE_SORTET[diFor2];
                        ayAT_INTERFACE_SORTET[diFor2]       := ayAT_INTERFACE_SORTET[diFor2 + 1];
                        ayAT_INTERFACE_SORTET[diFor2 + 1]   := ITF_AT_Temp;                                                
					END_IF;
				END_IF;
            END_IF;       
        END_FOR;      
    END_FOR;     
// 2 = Sort Vendor Name    
ELSIF uiSort = 2 THEN
    FOR diFor1 := LOWER_BOUND(ayAT_INTERFACE_SORTET,1) TO diMaxSort DO 
        FOR diFor2 := LOWER_BOUND(ayAT_INTERFACE_SORTET,1) TO diMaxSort -1 DO 
            IF ayAT_INTERFACE_SORTET[diFor2] <> 0 AND ayAT_INTERFACE_SORTET[diFor2 + 1] <> 0 THEN
                iBigger := fcGetBigerStringValue(ayAT_INTERFACE_SORTET[diFor2].proGetVendorDesignation,ayAT_INTERFACE_SORTET[diFor2 + 1].proGetVendorDesignation);
                IF iBigger = 1 THEN
                    ITF_AT_Temp                         := ayAT_INTERFACE_SORTET[diFor2];
                    ayAT_INTERFACE_SORTET[diFor2]       := ayAT_INTERFACE_SORTET[diFor2 + 1];
                    ayAT_INTERFACE_SORTET[diFor2 + 1]   := ITF_AT_Temp;                                            
                END_IF;
            END_IF;       
        END_FOR;      
    END_FOR;
// 3 & 4 = Sort State  
ELSIF uiSort = 3 OR uiSort = 4 THEN
    FOR diFor1 := LOWER_BOUND(ayAT_INTERFACE_SORTET,1) TO diMaxSort DO 
        FOR diFor2 := LOWER_BOUND(ayAT_INTERFACE_SORTET,1) TO diMaxSort -1 DO 
            IF ayAT_INTERFACE_SORTET[diFor2] <> 0 AND ayAT_INTERFACE_SORTET[diFor2 + 1] <> 0 THEN
                IF ayAT_INTERFACE_SORTET[diFor2].proIsError < ayAT_INTERFACE_SORTET[diFor2 + 1].proIsError THEN
                    ITF_AT_Temp                         := ayAT_INTERFACE_SORTET[diFor2];
                    ayAT_INTERFACE_SORTET[diFor2]       := ayAT_INTERFACE_SORTET[diFor2 + 1];
                    ayAT_INTERFACE_SORTET[diFor2 + 1]   := ITF_AT_Temp;    
                ELSIF NOT ayAT_INTERFACE_SORTET[diFor2].proIsError THEN
                    IF ayAT_INTERFACE_SORTET[diFor2].proIsWarning < ayAT_INTERFACE_SORTET[diFor2 + 1].proIsWarning THEN
                        ITF_AT_Temp                         := ayAT_INTERFACE_SORTET[diFor2];
                        ayAT_INTERFACE_SORTET[diFor2]       := ayAT_INTERFACE_SORTET[diFor2 + 1];
                        ayAT_INTERFACE_SORTET[diFor2 + 1]   := ITF_AT_Temp;    
                    ELSIF ayAT_INTERFACE_SORTET[diFor2].proIsEnabled < ayAT_INTERFACE_SORTET[diFor2 + 1].proIsEnabled THEN
                        ITF_AT_Temp                         := ayAT_INTERFACE_SORTET[diFor2];
                        ayAT_INTERFACE_SORTET[diFor2]       := ayAT_INTERFACE_SORTET[diFor2 + 1];
                        ayAT_INTERFACE_SORTET[diFor2 + 1]   := ITF_AT_Temp; 
                    ELSIF ayAT_INTERFACE_SORTET[diFor2].proIsWarning AND ayAT_INTERFACE_SORTET[diFor2 + 1].proIsWarning THEN
                        IF ayAT_INTERFACE_SORTET[diFor2].proRevisionSwitchOk > ayAT_INTERFACE_SORTET[diFor2 + 1].proRevisionSwitchOk THEN         
                            ITF_AT_Temp                         := ayAT_INTERFACE_SORTET[diFor2];
                            ayAT_INTERFACE_SORTET[diFor2]       := ayAT_INTERFACE_SORTET[diFor2 + 1];
                            ayAT_INTERFACE_SORTET[diFor2 + 1]   := ITF_AT_Temp; 
                        END_IF;       
                    END_IF;                                                       
                END_IF;
            END_IF;       
        END_FOR;      
    END_FOR;    
// 5 = Sort Stellwert Y   
ELSIF uiSort = 5 THEN
    FOR diFor1 := LOWER_BOUND(ayAT_INTERFACE_SORTET,1) TO diMaxSort DO 
        FOR diFor2 := LOWER_BOUND(ayAT_INTERFACE_SORTET,1) TO diMaxSort -1 DO 
            IF ayAT_INTERFACE_SORTET[diFor2] <> 0 AND ayAT_INTERFACE_SORTET[diFor2 + 1] <> 0 THEN
                IF ayAT_INTERFACE_SORTET[diFor2].proOnY < ayAT_INTERFACE_SORTET[diFor2 + 1].proOnY THEN
                    ITF_AT_Temp                         := ayAT_INTERFACE_SORTET[diFor2];
                    ayAT_INTERFACE_SORTET[diFor2]       := ayAT_INTERFACE_SORTET[diFor2 + 1];
                    ayAT_INTERFACE_SORTET[diFor2 + 1]   := ITF_AT_Temp;                                            
                END_IF;
            END_IF;       
        END_FOR;      
    END_FOR; 
// 6 = Sort Befehlt AUF   
ELSIF uiSort = 6 THEN
    FOR diFor1 := LOWER_BOUND(ayAT_INTERFACE_SORTET,1) TO diMaxSort DO 
        FOR diFor2 := LOWER_BOUND(ayAT_INTERFACE_SORTET,1) TO diMaxSort -1 DO 
            IF ayAT_INTERFACE_SORTET[diFor2] <> 0 AND ayAT_INTERFACE_SORTET[diFor2 + 1] <> 0 THEN
                IF ayAT_INTERFACE_SORTET[diFor2].proOnAuf < ayAT_INTERFACE_SORTET[diFor2 + 1].proOnAuf THEN
                    ITF_AT_Temp                         := ayAT_INTERFACE_SORTET[diFor2];
                    ayAT_INTERFACE_SORTET[diFor2]       := ayAT_INTERFACE_SORTET[diFor2 + 1];
                    ayAT_INTERFACE_SORTET[diFor2 + 1]   := ITF_AT_Temp;                                            
                END_IF;
            END_IF;       
        END_FOR;      
    END_FOR;   
// 7 = Sort Befehl ZU   
ELSIF uiSort = 7 THEN
    FOR diFor1 := LOWER_BOUND(ayAT_INTERFACE_SORTET,1) TO diMaxSort DO 
        FOR diFor2 := LOWER_BOUND(ayAT_INTERFACE_SORTET,1) TO diMaxSort -1 DO 
            IF ayAT_INTERFACE_SORTET[diFor2] <> 0 AND ayAT_INTERFACE_SORTET[diFor2 + 1] <> 0 THEN
                IF ayAT_INTERFACE_SORTET[diFor2].proOnZu < ayAT_INTERFACE_SORTET[diFor2 + 1].proOnZu THEN
                    ITF_AT_Temp                         := ayAT_INTERFACE_SORTET[diFor2];
                    ayAT_INTERFACE_SORTET[diFor2]       := ayAT_INTERFACE_SORTET[diFor2 + 1];
                    ayAT_INTERFACE_SORTET[diFor2 + 1]   := ITF_AT_Temp;                                            
                END_IF;
            END_IF;       
        END_FOR;      
    END_FOR;   
ELSE
    uiSort := 0;     
END_IF; 
IF uiSort = 0 AND stSearch = '' THEN
    xIsSortet := FALSE;  
ELSE
    xIsSortet := TRUE;  
END_IF
END_METHOD

PROPERTY proMin : INT
GET
proMin := 1;
END_GET
END_PROPERTY

PROPERTY proMax : UINT
GET
IF xIsSortet THEN
    proMax := LIMIT(0,TO_UINT(diMaxSort),65535);    
ELSE
    proMax := LIMIT(0,TO_UINT(diMax),65535);    
END_IF
END_GET
END_PROPERTY

PROPERTY proayStellAntriebTabelle : ARRAY[1..Parameter.iMaxStellAntrieb] OF ITF_STELLANTRIEB_TABELLE_INFO
GET
VAR
    diFor   :   DINT;
END_VAR
IF xIsSortet THEN
    FOR diFor := LOWER_BOUND(proayStellAntriebTabelle,1) TO UPPER_BOUND(proayStellAntriebTabelle,1) DO
        __QUERYINTERFACE(ayAT_INTERFACE_SORTET[diFor],proayStellAntriebTabelle[diFor]);   
	END_FOR
ELSE
    FOR diFor := LOWER_BOUND(proayStellAntriebTabelle,1) TO UPPER_BOUND(proayStellAntriebTabelle,1) DO
        __QUERYINTERFACE(ayAT_INTERFACE[diFor],proayStellAntriebTabelle[diFor]);   
	END_FOR
END_IF;
END_GET
END_PROPERTY

PROPERTY proMissedBuffer : DINT
GET
proMissedBuffer := diMissedBuffer;
END_GET
END_PROPERTY

PROPERTY proBufferError : BOOL
GET
proBufferError := xBufferError;
END_GET
END_PROPERTY

PROPERTY proayStellAntrieb : ARRAY[1..Parameter.iMaxStellAntrieb] OF ITF_STELLANTRIEB
GET
VAR
    diFor   :   DINT;
END_VAR
IF xIsSortet THEN
    proayStellAntrieb := ayAT_INTERFACE_SORTET;
ELSE
    proayStellAntrieb := ayAT_INTERFACE;
END_IF;
END_GET
END_PROPERTY

METHOD metGetStellAntriebITF : ITF_STELLANTRIEB
VAR_INPUT
    iPos    :   INT;
END_VAR
IF TO_DINT(iPos) >= LOWER_BOUND(ayAT_INTERFACE,1) AND TO_DINT(iPos) <= UPPER_BOUND(ayAT_INTERFACE,1) THEN
    IF xIsSortet THEN
        metGetStellAntriebITF := ayAT_INTERFACE_SORTET[iPos];       
    ELSE
        metGetStellAntriebITF := ayAT_INTERFACE[iPos];       
	END_IF   
END_IF
END_METHOD

END_FUNCTION_BLOCK

// 21 Interface/ITF_STELLANTRIEB_COLLECTOR
INTERFACE ITF_STELLANTRIEB_COLLECTOR

METHOD metSortArray
VAR_INPUT
    stSearch    :   STRING;
    uiSort      :   UINT;
END_VAR
END_METHOD

PROPERTY proayStellAntriebTabelle : ARRAY[1..Parameter.iMaxStellAntrieb] OF ITF_STELLANTRIEB_TABELLE_INFO
GET
END_GET
END_PROPERTY

PROPERTY proMax : UINT
GET
END_GET
END_PROPERTY

PROPERTY proMin : INT
GET
END_GET
END_PROPERTY

PROPERTY proBufferError : BOOL
GET
END_GET
END_PROPERTY

PROPERTY proMissedBuffer : DINT
GET
END_GET
END_PROPERTY

METHOD metGetStellAntriebITF : ITF_STELLANTRIEB
VAR_INPUT
    iPos    :   INT;
END_VAR
END_METHOD

END_INTERFACE

// 30 Program Organization Units/fcGetBigerStringValue
FUNCTION fcGetBigerStringValue : INT
VAR_INPUT
    st1     :   STRING(255);
    st2     :   STRING(255);
END_VAR
VAR
    diFor: DINT;
    diMax: DINT;
END_VAR

IF LEN(st1) > LEN(st2) THEN
    diMax := LEN(st2); 
    fcGetBigerStringValue := 1;
ELSIF LEN(st1) < LEN(st2) THEN
    diMax := LEN(st1);
    fcGetBigerStringValue := 2;     
ELSE
    diMax := LEN(st1);    
END_IF;
FOR diFor := 0 TO  diMax DO
    IF st1[diFor] > st2[diFor] THEN
        fcGetBigerStringValue := 1;  
        EXIT; 
    ELSIF st1[diFor] < st2[diFor] THEN
        fcGetBigerStringValue := 2;  
        EXIT;
    END_IF;
END_FOR;

END_FUNCTION

// 30 Program Organization Units/fcCheckQuerryReturnIcon
FUNCTION fcCheckQuerryReturnIcon : BOOL
VAR_INPUT
	_ITF_In			:	ITF_STELLANTRIEB;
	_uiIconNr_In	:	UINT;
END_VAR

IF __QUERYINTERFACE(_ITF_In,_ITF_In) THEN	
	fcCheckQuerryReturnIcon := TRUE;	
	_ITF_In.proValveIcon := _uiIconNr_In;
ELSE
	fcCheckQuerryReturnIcon := FALSE;	
END_IF

END_FUNCTION

// 30 Program Organization Units/Visu/fcValveAnimation
FUNCTION fcValveAnimation : INT
VAR_INPUT
	rProzent	:	REAL;
	xInvert		:	BOOL;
END_VAR
VAR
END_VAR

IF xInvert THEN
	fcValveAnimation := TO_INT(LIMIT(0,(100-rProzent)*10,1000));
ELSE
	fcValveAnimation := TO_INT(LIMIT(0,rProzent * 10,1000));
END_IF

END_FUNCTION

// 40 Visualizations/COLLECTOR/StellAntrieb_Collector
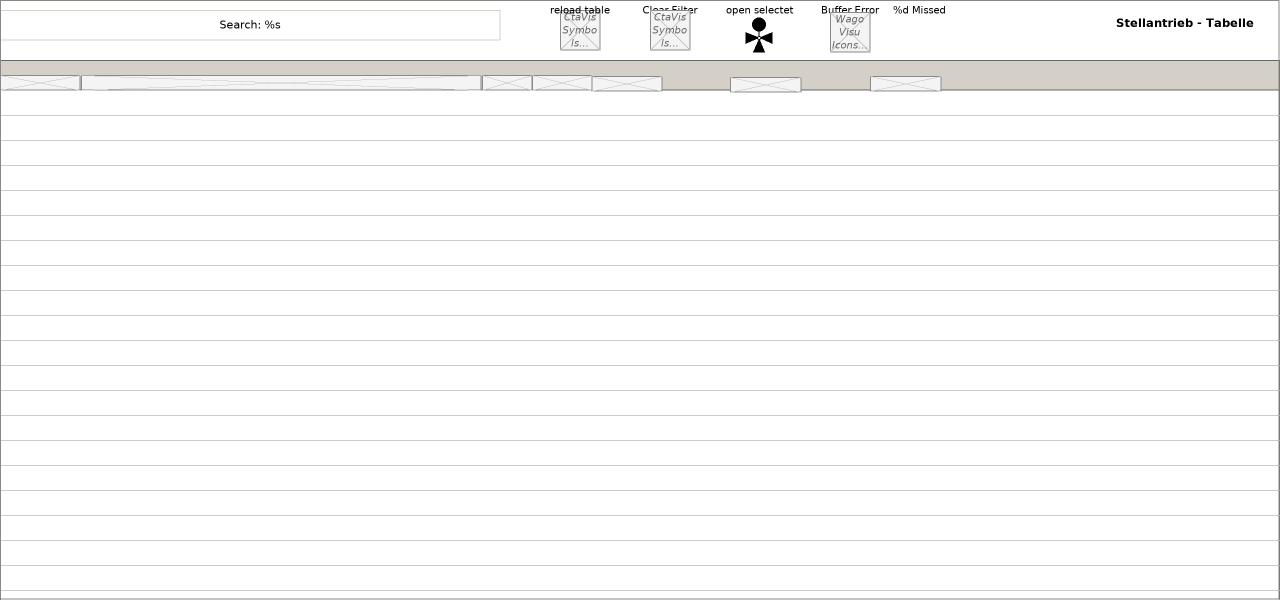
VISUALIZATION StellAntrieb_Collector  // 1280x600
    Frame (0,0 1280x600), invisible if: NOT GVL_StellAntrieb.xValidData
        shows StellAntrieb_Collector_TEMP(ayStellAntriebTabellenInfo := GVL_StellAntrieb.fbStellAntrieb_Collector.proayStellAntriebTabelle, uiMax := GVL_StellAntrieb.fbStellAntrieb_Collector.proMax, ITF_STELLANTRIEB_COLLECTOR := GVL_StellAntrieb.fbStellAntrieb_Collector)
END_VISUALIZATION

// 40 Visualizations/COLLECTOR/Help Funktionen/SelSort
VISUALIZATION SelSort  // 15x30
VAR_IN_OUT
	uiSel               :   UINT;
END_VAR
VAR_INPUT
    stSearch            :   STRING;    
    ITF_STELLANTRIEB_COLLECTOR    : ITF_STELLANTRIEB_COLLECTOR;
END_VAR
VAR_INPUT CONSTANT
    uiValue             :   UINT;
END_VAR
    Frame (0,15 15x15), invisible if: uiValue <> uiSel
        shows SortPfeil()
    Rectangle (0,0 15x30)
        OnMouseClick: execute {
            IF uiSel <> uiValue THEN
                uiSel   := uiValue;
            ELSE
                uiSel   := 0;
            END_IF
            ITF_STELLANTRIEB_COLLECTOR.metSortArray(stSearch,uiSel);
        }
END_VISUALIZATION

// 40 Visualizations/COLLECTOR/StellAntrieb_Collector_TEMP
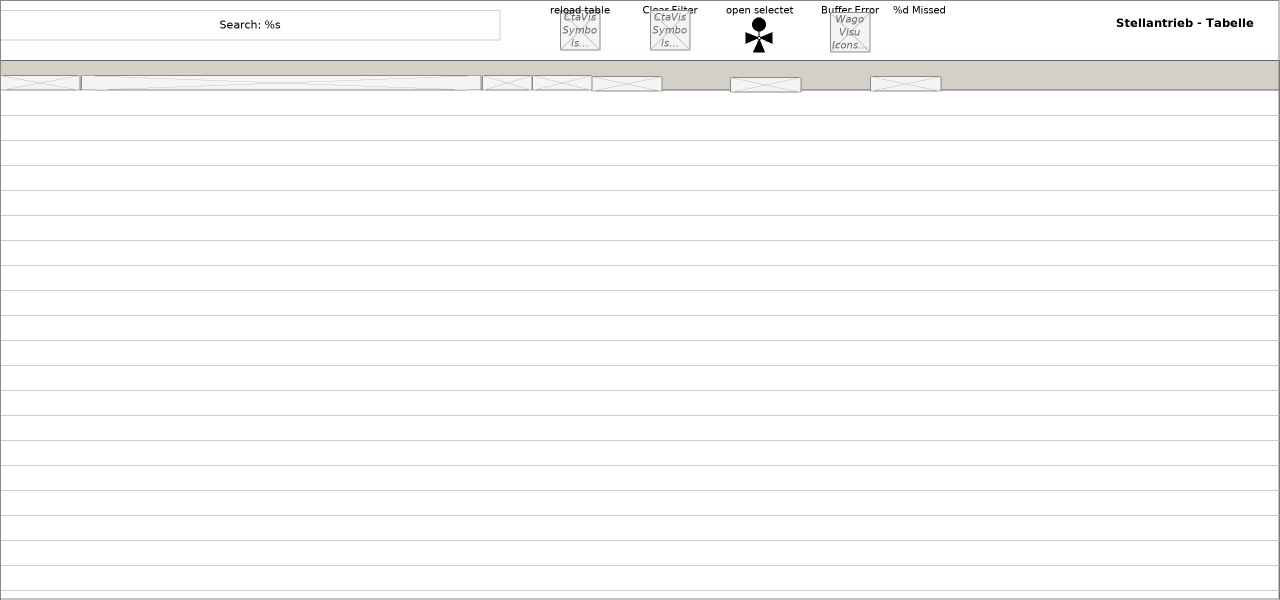
VISUALIZATION StellAntrieb_Collector_TEMP  // 1280x600
VAR_INPUT
	ayStellAntriebTabellenInfo  : 	ARRAY[1..Parameter.iMaxStellAntrieb] OF ITF_STELLANTRIEB_TABELLE_INFO;
    uiMax                   	: 	UINT;
    ITF_STELLANTRIEB_COLLECTOR        	:	ITF_STELLANTRIEB_COLLECTOR;
END_VAR
VAR
    iZeile                  	:   INT;
    stSearch               		:   STRING;
    uiSort                  	:   UINT;
    xReadySearch           		:   BOOL;
END_VAR
    Table (0,60 1280x541), data array: ayStellAntriebTabellenInfo
        p1128707560: uiMax
        p1014161805: Parameter.iMaxStellAntrieb - 1 + 1
        p1137915858: iZeile
        p3136911649: ayStellAntriebTabellenInfo[INDEX].proGetInstancePath
        p797552052: ayStellAntriebTabellenInfo[INDEX].proSetInstancePath
        p400160035: ayStellAntriebTabellenInfo[INDEX].proNoBmkInList
        p2319025000: ayStellAntriebTabellenInfo[INDEX].proGetObjectId
        p4242324053: ayStellAntriebTabellenInfo[INDEX].proGetCustomerDesignation
        p3863566920: ayStellAntriebTabellenInfo[INDEX].proGetBMK
        p1933151965: ayStellAntriebTabellenInfo[INDEX].proStateSymbol
        p1739542657: ayStellAntriebTabellenInfo[INDEX].proGetAKS
        p511219082: Vendor designation
        p1892666644: ayStellAntriebTabellenInfo[INDEX].proGetVendorDesignation
        p2170511999: ayStellAntriebTabellenInfo[INDEX].proEnSymbol
        p4092479075: Enabled
        p338671338: ayStellAntriebTabellenInfo[INDEX].proRükIsOpen
        p746581629: ayStellAntriebTabellenInfo[INDEX].proOnAuf
        p1757482276: Open OUT
        p1218418051: ayStellAntriebTabellenInfo[INDEX].proIsOnY
        p505689113: Y IN
        p3723444502: ayStellAntriebTabellenInfo[INDEX].proOnY
        p2237128397: Y OUT
        p7306298: ayStellAntriebTabellenInfo[INDEX].proRükIsClosed
        p516019884: Closed IN
        p2501879983: ayStellAntriebTabellenInfo[INDEX].proOnZu
        p2243050616: Close OUT
        p4088588272: Open IN
    Textfield (0,10 500x30), "Search: %s", text variable: stSearch
        OnMouseClick: write the text variable via Default
        OnMouseClick: execute { xReadySearch := TRUE; }
    Image (560,10 40x40), invisible if: NOT xReadySearch, image: CtaVisSymbols.ImagePool.refresh_solo_black
        OnMouseClick: execute { ITF_STELLANTRIEB_COLLECTOR.metSortArray(stSearch,uiSort); xReadySearch := FALSE; }
    Label (540,5 80x10), "reload table", invisible if: NOT xReadySearch
    Label (720,5 80x10), "open selectet", invisible if: TO_DINT(iZeile) < LOWER_BOUND(ayStellAntriebTabellenInfo,1) OR TO_DINT(iZeile) > UPPER_BOUND(ayStellAntriebTabellenInfo,1)
    Label (630,5 80x10), "Clear Filter", invisible if: stSearch = '' AND uiSort = 0
    Image (650,10 40x40), invisible if: stSearch = '' AND uiSort = 0, image: CtaVisSymbols.ImagePool.close_solo_black
        OnMouseClick: execute {
            stSearch := '';
            uiSort   := 0;
            ITF_STELLANTRIEB_COLLECTOR.metSortArray(stSearch,uiSort);
            xReadySearch := FALSE;
        }
    Label (1095,8 180x30), "Stellantrieb - Tabelle"
    Label (810,5 80x10), "Buffer Error", invisible if: NOT ITF_STELLANTRIEB_COLLECTOR.proBufferError
    Image (830,12 40x40), invisible if: NOT ITF_STELLANTRIEB_COLLECTOR.proBufferError, image: WagoVisuIcons.WagoIcons.4
    Textfield (890,5 100x10), "%d Missed", text variable: ITF_STELLANTRIEB_COLLECTOR.proMissedBuffer, invisible if: NOT ITF_STELLANTRIEB_COLLECTOR.proBufferError
    Frame (741,16 40x40), invisible if: TO_DINT(iZeile) < LOWER_BOUND(ayStellAntriebTabellenInfo,1) OR TO_DINT(iZeile) > UPPER_BOUND(ayStellAntriebTabellenInfo,1)
        shows StellAntrieb_Icon_StellAntrieb()
        OnMouseClick:  Dialog=StellAntrieb_POPUP, Parameters={ITF_STELLANTRIEBIN: ITF_STELLANTRIEB_COLLECTOR.metGetStellAntriebITF(iZeile), uiPopUpGruppe: 0}, OpenModal=True, OpenCentered=True
    Frame (870,61 71x30)
        shows SelSort(uiSel := uiSort, stSearch := stSearch, ITF_STELLANTRIEB_COLLECTOR := ITF_STELLANTRIEB_COLLECTOR, uiValue := 7)
    Frame (730,62 71x30)
        shows SelSort(uiSel := uiSort, stSearch := stSearch, ITF_STELLANTRIEB_COLLECTOR := ITF_STELLANTRIEB_COLLECTOR, uiValue := 6)
    Frame (591,61 71x30)
        shows SelSort(uiSel := uiSort, stSearch := stSearch, ITF_STELLANTRIEB_COLLECTOR := ITF_STELLANTRIEB_COLLECTOR, uiValue := 5)
    Frame (532,60 60x30)
        shows SelSort(uiSel := uiSort, stSearch := stSearch, ITF_STELLANTRIEB_COLLECTOR := ITF_STELLANTRIEB_COLLECTOR, uiValue := 4)
    Frame (482,60 50x30)
        shows SelSort(uiSel := uiSort, stSearch := stSearch, ITF_STELLANTRIEB_COLLECTOR := ITF_STELLANTRIEB_COLLECTOR, uiValue := 3)
    Frame (81,60 400x30)
        shows SelSort(uiSel := uiSort, stSearch := stSearch, ITF_STELLANTRIEB_COLLECTOR := ITF_STELLANTRIEB_COLLECTOR, uiValue := 2)
    Frame (0,60 80x30)
        shows SelSort(uiSel := uiSort, stSearch := stSearch, ITF_STELLANTRIEB_COLLECTOR := ITF_STELLANTRIEB_COLLECTOR, uiValue := 1)
END_VISUALIZATION

// 40 Visualizations/COLLECTOR/Help Funktionen/SortPfeil
VISUALIZATION SortPfeil  // 15x15
    Image (0,0 15x15), image: CtaVisSymbols.ImagePool.arrow-down_solo_black
END_VISUALIZATION

// 40 Visualizations/POPUP/StellAntrieb_POPUP
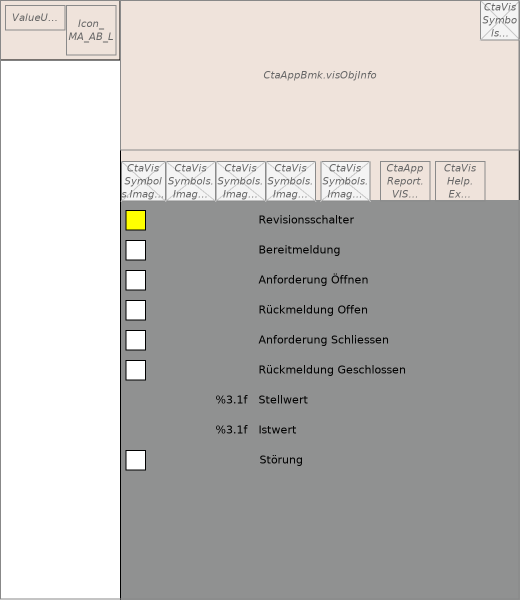
VISUALIZATION StellAntrieb_POPUP  // 520x600
VAR_INPUT
    ITF_STELLANTRIEBIN  :   ITF_STELLANTRIEB;
	stExklParameter		:	STRING[40];
	uiPopUpGruppe		: 	UINT;
END_VAR
    Rectangle (0,0 120x60)
    Rectangle (120,0 400x600)
    Frame (120,0 400x150)
        shows CtaAppBmk.visObjInfo(ITF_BMK_IN := ITF_STELLANTRIEBIN)
    Image (480,0 40x40), image: CtaVisSymbols.ImagePool.close_solo_black
        OnMouseClick:  Dialog=StellAntrieb_POPUP, Result=None, NumpadKeypadSet=True
    Frame (121,200 399x400), frame switch variable: uiPopUpGruppe
        shows StellAntrieb_OVERVIEW(ITF_STELLANTRIEBIN := ITF_STELLANTRIEBIN)
        shows StellAntrieb_MANUAL(ITF_STELLANTRIEBIN := ITF_STELLANTRIEBIN)
        shows StellAntrieb_PARAMETER(ITF_STELLANTRIEBIN := ITF_STELLANTRIEBIN)
        shows StellAntrieb_IO(ITF_STELLANTRIEBIN := ITF_STELLANTRIEBIN)
        shows StellAntrieb_BUS(ITF_STELLANTRIEBIN := ITF_STELLANTRIEBIN)
        shows StellAntrieb_REPORTS(ITF_STELLANTRIEBIN := ITF_STELLANTRIEBIN)
    Frame (121,161 399x40)
        shows StellAntrieb_PopUpListe(uiPopUpGruppe := uiPopUpGruppe, xHand := ITF_STELLANTRIEBIN.proIsHandOnOrOff, xHandOff := ITF_STELLANTRIEBIN.proHandOff, ITF_REPORTMANAGER_IN := ITF_STELLANTRIEBIN.proITF_REPORTMANAGER, stExklParameter := stExklParameter)
        pReferences[0]: AnzError=ITF_STELLANTRIEBIN.proAnzError, AnzWarning=ITF_STELLANTRIEBIN.proAnzWarning
    Frame (5,5 110x50), input disabled if: TRUE, frame switch variable: ITF_STELLANTRIEBIN.proValveIcon
        shows StellAntrieb_MA_Valve_AB_Left_Txt_L_Above(ITF_STELLANTRIEB_IN := ITF_STELLANTRIEBIN, stExklParameter := stExklParameter)
        shows StellAntrieb_MA_Valve_AB_Right_Txt_L_Above(ITF_STELLANTRIEB_IN := ITF_STELLANTRIEBIN, stExklParameter := stExklParameter)
        shows StellAntrieb_MA_Valve_Flow_Txt_L_Above(ITF_STELLANTRIEB_IN := ITF_STELLANTRIEBIN, stExklParameter := stExklParameter)
        shows StellAntrieb_MA_Valve_Mix_Txt_L_Above(ITF_STELLANTRIEB_IN := ITF_STELLANTRIEBIN, stExklParameter := stExklParameter)
        shows StellAntrieb_MB_Valve_AB_Left_Txt_L_Below(ITF_STELLANTRIEB_IN := ITF_STELLANTRIEBIN, stExklParameter := stExklParameter)
        shows StellAntrieb_MB_Valve_AB_Right_Txt_L_Below(ITF_STELLANTRIEB_IN := ITF_STELLANTRIEBIN, stExklParameter := stExklParameter)
        shows StellAntrieb_MB_Valve_Flow_Txt_L_Below(ITF_STELLANTRIEB_IN := ITF_STELLANTRIEBIN, stExklParameter := stExklParameter)
        shows StellAntrieb_MB_Valve_Mix_Txt_L_Below(ITF_STELLANTRIEB_IN := ITF_STELLANTRIEBIN, stExklParameter := stExklParameter)
        shows StellAntrieb_ML_Valve_AB_Down_Txt_L_Above(ITF_STELLANTRIEB_IN := ITF_STELLANTRIEBIN, stExklParameter := stExklParameter)
        shows StellAntrieb_ML_Valve_AB_Down_Txt_L_Below(ITF_STELLANTRIEB_IN := ITF_STELLANTRIEBIN, stExklParameter := stExklParameter)
        shows StellAntrieb_ML_Valve_AB_Up_Txt_L_Above(ITF_STELLANTRIEB_IN := ITF_STELLANTRIEBIN, stExklParameter := stExklParameter)
        shows StellAntrieb_ML_Valve_AB_Up_Txt_L_Below(ITF_STELLANTRIEB_IN := ITF_STELLANTRIEBIN, stExklParameter := stExklParameter)
        shows StellAntrieb_ML_Valve_Flow_Txt_L_Above(ITF_STELLANTRIEB_IN := ITF_STELLANTRIEBIN, stExklParameter := stExklParameter)
        shows StellAntrieb_ML_Valve_Flow_Txt_L_Below(ITF_STELLANTRIEB_IN := ITF_STELLANTRIEBIN, stExklParameter := stExklParameter)
        shows StellAntrieb_ML_Valve_Mix_Txt_L_Above(ITF_STELLANTRIEB_IN := ITF_STELLANTRIEBIN, stExklParameter := stExklParameter)
        shows StellAntrieb_ML_Valve_Mix_Txt_L_Below(ITF_STELLANTRIEB_IN := ITF_STELLANTRIEBIN, stExklParameter := stExklParameter)
        shows StellAntrieb_MA_Valve_AB_Left_Txt_R_Above(ITF_STELLANTRIEB_IN := ITF_STELLANTRIEBIN, stExklParameter := stExklParameter)
        shows StellAntrieb_MA_Valve_AB_Right_Txt_R_Above(ITF_STELLANTRIEB_IN := ITF_STELLANTRIEBIN, stExklParameter := stExklParameter)
        shows StellAntrieb_MA_Valve_Flow_Txt_R_Above(ITF_STELLANTRIEB_IN := ITF_STELLANTRIEBIN, stExklParameter := stExklParameter)
        shows StellAntrieb_MA_Valve_Mix_Txt_R_Above(ITF_STELLANTRIEB_IN := ITF_STELLANTRIEBIN, stExklParameter := stExklParameter)
        shows StellAntrieb_MB_Valve_AB_Left_Txt_R_Below(ITF_STELLANTRIEB_IN := ITF_STELLANTRIEBIN, stExklParameter := stExklParameter)
        shows StellAntrieb_MB_Valve_AB_Right_Txt_R_Below(ITF_STELLANTRIEB_IN := ITF_STELLANTRIEBIN, stExklParameter := stExklParameter)
        shows StellAntrieb_MB_Valve_Flow_Txt_R_Below(ITF_STELLANTRIEB_IN := ITF_STELLANTRIEBIN, stExklParameter := stExklParameter)
        shows StellAntrieb_MB_Valve_Mix_Txt_R_Below(ITF_STELLANTRIEB_IN := ITF_STELLANTRIEBIN, stExklParameter := stExklParameter)
        shows StellAntrieb_MR_Valve_AB_Down_Txt_R_Above(ITF_STELLANTRIEB_IN := ITF_STELLANTRIEBIN, stExklParameter := stExklParameter)
        shows StellAntrieb_MR_Valve_AB_Down_Txt_R_Below(ITF_STELLANTRIEB_IN := ITF_STELLANTRIEBIN, stExklParameter := stExklParameter)
        shows StellAntrieb_MR_Valve_AB_Up_Txt_R_Above(ITF_STELLANTRIEB_IN := ITF_STELLANTRIEBIN, stExklParameter := stExklParameter)
        shows StellAntrieb_MR_Valve_AB_Up_Txt_R_Below(ITF_STELLANTRIEB_IN := ITF_STELLANTRIEBIN, stExklParameter := stExklParameter)
        shows StellAntrieb_MR_Valve_Flow_Txt_R_Above(ITF_STELLANTRIEB_IN := ITF_STELLANTRIEBIN, stExklParameter := stExklParameter)
        shows StellAntrieb_MR_Valve_Flow_Txt_R_Below(ITF_STELLANTRIEB_IN := ITF_STELLANTRIEBIN, stExklParameter := stExklParameter)
        shows StellAntrieb_MR_Valve_Mix_Txt_R_Above(ITF_STELLANTRIEB_IN := ITF_STELLANTRIEBIN, stExklParameter := stExklParameter)
        shows StellAntrieb_MR_Valve_Mix_Txt_R_Below(ITF_STELLANTRIEB_IN := ITF_STELLANTRIEBIN, stExklParameter := stExklParameter)
        shows S_AT_MR_Valve_AB_Up_Txt_R_Above()
        shows S_AT_MR_Valve_AB_Up_Txt_R_Below()
        shows S_AT_MR_Flap_Txt_R_Above()
        shows S_AT_MR_Flap_Txt_R_Below()
        shows S_AT_MR_Valve_Flow_Txt_R_Above()
        shows S_AT_MR_Valve_Flow_Txt_R_Below()
        shows S_AT_MR_Valve_Mix_Txt_R_Above()
        shows S_AT_MR_Valve_Mix_Txt_R_Below()
END_VISUALIZATION

// 40 Visualizations/POPUP/StellAntrieb_PopUpListe
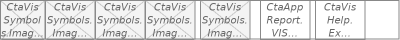
VISUALIZATION StellAntrieb_PopUpListe  // 400x40
VAR_IN_OUT
	uiPopUpGruppe : UINT;
END_VAR
VAR_INPUT
    xHand           		: BOOL;
    xHandOff        		: BOOL;
    ITF_REPORTMANAGER_IN    : CtaAppReport.ITF_REPORTMANAGER;
    stExklParameter     	: STRING [40];
END_VAR
    Rectangle (100,0 40x40), colour toggle: uiPopUpGruppe = 2
        OnMouseDown: execute { uiPopUpGruppe := 2; }
    Rectangle (50,0 40x40), colour toggle: uiPopUpGruppe = 1
        OnMouseDown: execute { uiPopUpGruppe := 1; }
    Rectangle (0,0 40x40), colour toggle: uiPopUpGruppe = 0
        OnMouseDown: execute { uiPopUpGruppe := 0; }
    Image (0,0 45x40), image: CtaVisSymbols.ImagePool.eye
        OnMouseDown: execute { uiPopUpGruppe := 0; }
    Image (45,0 50x40), image: CtaVisSymbols.ImagePool.front_hand_Black
        OnMouseDown: execute { uiPopUpGruppe := 1; }
    Image (95,0 50x40), image: CtaVisSymbols.ImagePool.gear
        OnMouseDown: execute { uiPopUpGruppe := 2; }
    Image (45,0 50x40), invisible if: NOT xHand, image: CtaVisSymbols.ImagePool.front_hand_Yellow
        OnMouseDown: execute { uiPopUpGruppe := 1; }
    Rectangle (205,0 40x40), colour toggle: uiPopUpGruppe = 4
        OnMouseDown: execute { uiPopUpGruppe := 4; }
    Image (200,0 50x40), image: CtaVisSymbols.ImagePool.lan
        OnMouseDown: execute { uiPopUpGruppe := 4; }
    Image (45,0 50x40), invisible if: NOT xHandOff, image: CtaVisSymbols.ImagePool.front_hand_Yellow_Off
        OnMouseDown: execute { uiPopUpGruppe := 1; }
    Rectangle (150,0 40x40), colour toggle: uiPopUpGruppe = 3
        OnMouseDown: execute { uiPopUpGruppe := 3; }
    Image (145,0 50x40), image: CtaVisSymbols.ImagePool.dip-switch
        OnMouseDown: execute { uiPopUpGruppe := 3; }
    Rectangle (260,0 50x40), colour toggle: uiPopUpGruppe = 5
        OnMouseDown: execute { uiPopUpGruppe := 5; }
    Frame (260,0 50x40)
        shows CtaAppReport.VIS_ANZ_REPORTS_MODUL(ITF_REPORTMANAGER_IN := ITF_REPORTMANAGER_IN)
        OnMouseDown: execute { uiPopUpGruppe := 5; }
    Rectangle (315,0 50x40), colour toggle: uiPopUpGruppe = 6
        OnMouseDown: execute { uiPopUpGruppe := 6; }
    Frame (315,0 50x40)
        shows CtaVisHelp.ExkParameterSymbol(stExklParameter := stExklParameter)
END_VISUALIZATION

// 40 Visualizations/ICON/StellAntrieb_RIGHT/Motor_Right/Valve_AB_Down/Above/StellAntrieb_MR_Valve_AB_Down_RA_CheckQuerry
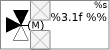
VISUALIZATION StellAntrieb_MR_Valve_AB_Down_RA_CheckQuerry  // 110x50
VAR_INPUT
    ITF_STELLANTRIEB_IN   	:   ITF_STELLANTRIEB;
	stExklParameter			:	STRING[40];
END_VAR
    Frame (0,0 110x50)
        shows StellAntrieb_MR_Valve_AB_Down_RA_CheckEnabled(ITF_STELLANTRIEB_IN := ITF_STELLANTRIEB_IN, stExklParameter := stExklParameter)
END_VISUALIZATION

// 40 Visualizations/ICON/StellAntrieb_RIGHT/Motor_Right/Valve_AB_Down/Above/StellAntrieb_MR_Valve_AB_Down_Txt_R_Above
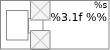
VISUALIZATION StellAntrieb_MR_Valve_AB_Down_Txt_R_Above  // 110x50
VAR_INPUT
    ITF_STELLANTRIEB_IN   	:   ITF_STELLANTRIEB;	
END_VAR
VAR_INPUT CONSTANT
	stExklParameter			:	STRING[40] := '';
END_VAR
VAR CONSTANT
	uiIconNr				: 	UINT := 24;
END_VAR
    Frame (0,0 110x50), invisible if: NOT fcCheckQuerryReturnIcon(_ITF_In := ITF_STELLANTRIEB_IN,_uiIconNr_In := uiIconNr)
        shows StellAntrieb_MR_Valve_AB_Down_RA_CheckQuerry(ITF_STELLANTRIEB_IN := ITF_STELLANTRIEB_IN, stExklParameter := stExklParameter)
        shows Icon()
END_VISUALIZATION

// 40 Visualizations/ICON/StellAntrieb_RIGHT/Motor_Right/Valve_AB_Down/Above/StellAntrieb_MR_Valve_AB_Down_RA_CheckEnabled
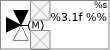
VISUALIZATION StellAntrieb_MR_Valve_AB_Down_RA_CheckEnabled  // 110x50
VAR_INPUT
    ITF_STELLANTRIEB_IN   	:   ITF_STELLANTRIEB;
	stExklParameter			:	STRING[40];
END_VAR
    Frame (0,0 50x50), invisible if: NOT ITF_STELLANTRIEB_IN.proIsEnabled
        shows Icon_MR_AB_Down(ITF_STELLANTRIEB_IN := ITF_STELLANTRIEB_IN)
    Frame (50,0 60x25), invisible if: NOT ITF_STELLANTRIEB_IN.proIsEnabled
        shows ValueUpDwn(ITF_STELLANTRIEB_IN := ITF_STELLANTRIEB_IN, uiTextAusrichtung := 4)
    Rectangle (0,0 110x50)
        OnMouseClick:  Dialog=StellAntrieb_POPUP, Parameters={stExklParameter: stExklParameter, ITF_STELLANTRIEBIN: ITF_STELLANTRIEB_IN, uiPopUpGruppe: 0}, OpenCentered=True
END_VISUALIZATION

// 40 Visualizations/ICON/StellAntrieb_BASE/Icons/Motor
VISUALIZATION Motor  // 15x15
VAR_INPUT
    ITF_STELLANTRIEB_IN   :   ITF_STELLANTRIEB;	
END_VAR
    Ellipse (0,0 15x15), "M", colour toggle: ITF_STELLANTRIEB_IN.proIsError
    Ellipse (0,0 15x15), "M", colour toggle: ITF_STELLANTRIEB_IN.proOn, invisible if: ITF_STELLANTRIEB_IN.proIsError
END_VISUALIZATION

// 40 Visualizations/POPUP/PARAMETER/StellAntrieb_PARAMETER
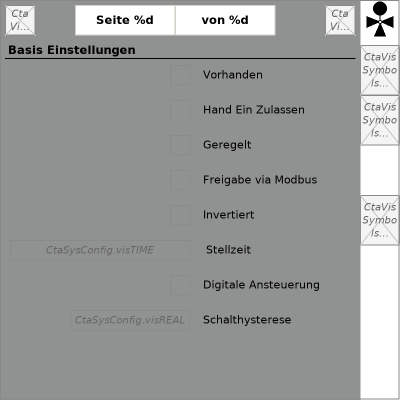
VISUALIZATION StellAntrieb_PARAMETER  // 400x400
VAR_INPUT
    ITF_STELLANTRIEBIN 	:	ITF_STELLANTRIEB;
END_VAR
VAR
    uiParameterGruppe : UINT;
END_VAR
    Image (145,122 150x30), image: ImagePool.Kreis
    Frame (360,0 40x300)
        shows StellAntrieb_ParameterListe(uiParameterGruppe := uiParameterGruppe)
    Frame (0,0 360x400), frame switch variable: uiParameterGruppe
        shows StellAntrieb_ParameterBase(ITF_STELLANTRIEBIN := ITF_STELLANTRIEBIN)
        shows StellAntrieb_ParameterFuses(ITF_STELLANTRIEBIN := ITF_STELLANTRIEBIN)
        shows StellAntrieb_ParameterIO(ITF_STELLANTRIEBIN := ITF_STELLANTRIEBIN)
        shows StellAntrieb_ParameterInfluxDb(ITF_STELLANTRIEBIN := ITF_STELLANTRIEBIN)
        shows S_AT_ParameterInfluxDb(ITF_Parameter := ITF_Parameter)
        pReferences[0]: ITF_Parameter=ITF_Parameter
        pReferences[1]: ITF_Parameter=ITF_Parameter
        pReferences[2]: ITF_Parameter=ITF_Parameter
        pReferences[3]: ITF_Parameter=ITF_Parameter
END_VISUALIZATION

// 40 Visualizations/POPUP/PARAMETER/StellAntrieb_ParameterListe
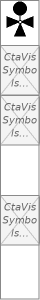
VISUALIZATION StellAntrieb_ParameterListe  // 40x300
VAR_IN_OUT
	uiParameterGruppe : UINT;
END_VAR
    Rectangle (0,0 39x40), colour toggle: uiParameterGruppe = 0
        OnMouseDown: execute { uiParameterGruppe := 0; }
    Frame (2,0 40x40)
        shows StellAntrieb_Icon_StellAntrieb()
        OnMouseDown: execute { uiParameterGruppe := 0; }
    Rectangle (0,100 39x40), colour toggle: uiParameterGruppe = 2
        OnMouseDown: execute { uiParameterGruppe := 2; }
    Rectangle (0,50 39x40), colour toggle: uiParameterGruppe = 1
        OnMouseDown: execute { uiParameterGruppe := 1; }
    Image (0,45 40x50), image: CtaVisSymbols.ImagePool.lightning-bolt-circle
        OnMouseDown: execute { uiParameterGruppe := 1; }
    Rectangle (0,200 39x40), colour toggle: uiParameterGruppe = 3
        OnMouseDown: execute { uiParameterGruppe := 3; }
    Image (0,195 40x50), image: CtaVisSymbols.ImagePool.sine-wave
        OnMouseDown: execute { uiParameterGruppe := 3; }
    Image (0,95 40x50), image: CtaVisSymbols.ImagePool.dip-switch
        OnMouseDown: execute { uiParameterGruppe := 2; }
END_VISUALIZATION

// 40 Visualizations/POPUP/MANUAL/StellAntrieb_MANUAL
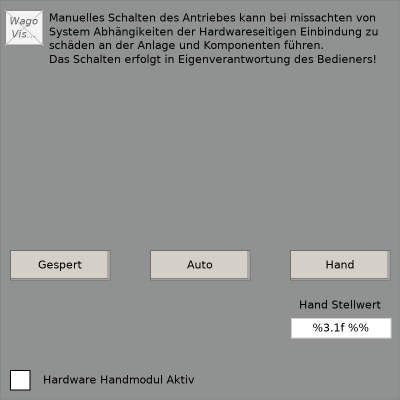
VISUALIZATION StellAntrieb_MANUAL  // 400x400
VAR_INPUT
    ITF_STELLANTRIEBIN    :   ITF_STELLANTRIEB;	
END_VAR
    Button (10,250 100x30), "Gespert", colour toggle: ITF_STELLANTRIEBIN.proHandOff, pressed state: ITF_STELLANTRIEBIN.proHandOff
        toggle ITF_STELLANTRIEBIN.proHandOff
    Button (290,250 100x30), "Hand", colour toggle: ITF_STELLANTRIEBIN.proHandOn, pressed state: ITF_STELLANTRIEBIN.proHandOn
        toggle ITF_STELLANTRIEBIN.proHandOn
    Button (150,250 100x30), "Auto", colour toggle: ITF_STELLANTRIEBIN.proAuto, pressed state: ITF_STELLANTRIEBIN.proAuto
        toggle ITF_STELLANTRIEBIN.proAuto
    Label (46,10 350x100), "Manuelles Schalten des Antriebes kann bei missachten von System Abhängikeiten der Hardwareseitigen Einbindung zu schäden an der Anlage und Komponenten führen. Das Schalten erfolgt in Eigenverantwortung des Bedieners!"
    Textfield (291,318 100x20), "%3.1f %%", text variable: ITF_STELLANTRIEBIN.proHandOnY, invisible if: NOT ITF_STELLANTRIEBIN.proIsRegulatet
        OnMouseClick: write the text variable via InputWithLimits, min 0, max 100, title 'Stellwert'
    Image (5,10 38x35), image: WagoVisuIcons.WagoIcons.2
    Label (290,295 100x20), "Hand Stellwert"
    Rectangle (10,370 20x20), colour toggle: ITF_STELLANTRIEBIN.proHardWareHandModulAktive, invisible if: NOT ITF_STELLANTRIEBIN.proHardWareHandModulAktive
    Label (40,370 200x20), "Hardware Handmodul Aktiv", invisible if: NOT ITF_STELLANTRIEBIN.proHardWareHandModulAktive
END_VISUALIZATION

// 40 Visualizations/POPUP/OVERVIEW/StellAntrieb_OVERVIEW
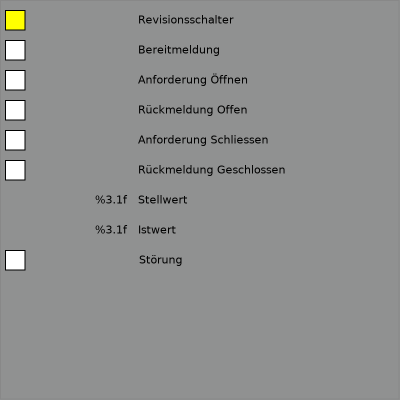
VISUALIZATION StellAntrieb_OVERVIEW  // 400x400
VAR_INPUT
    ITF_STELLANTRIEBIN    :   ITF_STELLANTRIEB;	
END_VAR
    Label (135,10 200x20), "Revisionsschalter"
    Label (135,40 200x20), "Bereitmeldung"
    Rectangle (5,10 20x20), colour toggle: ITF_STELLANTRIEBIN.proRevisionSwitchOk
    Rectangle (5,40 20x20), colour toggle: ITF_STELLANTRIEBIN.proIsReady
    Label (135,190 200x20), "Stellwert", invisible if: NOT ITF_STELLANTRIEBIN.proIsRegulatet
    Label (135,220 200x20), "Istwert", invisible if: NOT ITF_STELLANTRIEBIN.proIsRegulatet
    Textfield (30,190 100x20), "%3.1f", text variable: ITF_STELLANTRIEBIN.proOnY, invisible if: NOT ITF_STELLANTRIEBIN.proIsRegulatet
    Textfield (30,220 100x20), "%3.1f", text variable: ITF_STELLANTRIEBIN.proIsOnY, invisible if: NOT ITF_STELLANTRIEBIN.proIsRegulatet
    Rectangle (5,70 20x20), colour toggle: ITF_STELLANTRIEBIN.proOnAuf
    Label (135,70 200x20), "Anforderung Öffnen"
    Rectangle (5,100 20x20), colour toggle: ITF_STELLANTRIEBIN.proRükIsOpen, invisible if: ITF_STELLANTRIEBIN.proNotShowDI_RükIsOpen
    Label (135,100 200x20), "Rückmeldung Offen", invisible if: ITF_STELLANTRIEBIN.proNotShowDI_RükIsOpen
    Rectangle (5,130 20x20), colour toggle: ITF_STELLANTRIEBIN.proOnZu
    Label (135,130 200x20), "Anforderung Schliessen"
    Rectangle (5,160 20x20), colour toggle: ITF_STELLANTRIEBIN.proRükIsClosed, invisible if: ITF_STELLANTRIEBIN.proNotShowDI_RükIsClosed
    Label (135,160 200x20), "Rückmeldung Geschlossen", invisible if: ITF_STELLANTRIEBIN.proNotShowDI_RükIsClosed
    Rectangle (5,250 20x20), colour toggle: ITF_STELLANTRIEBIN.proIsError
    Label (136,250 200x20), "Störung"
END_VISUALIZATION

// 40 Visualizations/POPUP/BUS/StellAntrieb_BUS
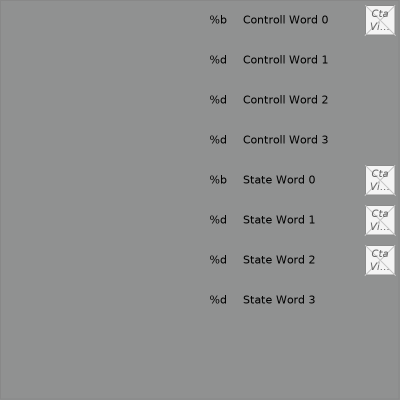
VISUALIZATION StellAntrieb_BUS  // 400x400
VAR_INPUT
    ITF_STELLANTRIEBIN    :   ITF_STELLANTRIEB;	
END_VAR
    Frame (100,0 300x350)
        shows StellAntrieb_BUS_CS(ITF_STELLANTRIEBIn := ITF_STELLANTRIEBIN, ayControllWord := ITF_STELLANTRIEBIN.proModbusControllWord, ayStateWord := ITF_STELLANTRIEBIN.proModbusStateWord)
END_VISUALIZATION

// 40 Visualizations/POPUP/BUS/StellAntrieb_BUS_SW0_Detail
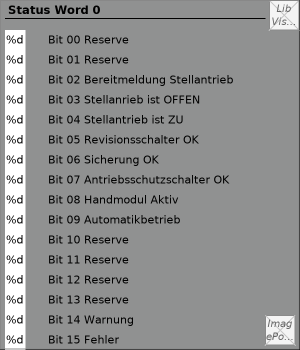
VISUALIZATION StellAntrieb_BUS_SW0_Detail  // 300x350
VAR_IN_OUT
    wDetail     :   WORD;
END_VAR
VAR_INPUT	
    ITF_STELLANTRIEBIN    :   ITF_STELLANTRIEB;
END_VAR
VAR_IN_OUT
    xShow       :   BOOL;
END_VAR
    Rectangle (0,0 300x350)
    Textfield (5,30 20x20), "%d", text variable: TO_WORD(wDetail.0), input disabled if: NOT ITF_STELLANTRIEBIn.proModbusTest
        OnMouseClick: execute { wDetail.0 := NOT wDetail.0; }
    Label (45,30 180x20), "Bit 00 Reserve"
    Textfield (5,50 20x20), "%d", text variable: TO_WORD(wDetail.1), input disabled if: NOT ITF_STELLANTRIEBIn.proModbusTest
        OnMouseClick: execute { wDetail.1 := NOT wDetail.1; }
    Label (45,50 180x20), "Bit 01 Reserve"
    Textfield (5,70 20x20), "%d", text variable: TO_WORD(wDetail.2), input disabled if: NOT ITF_STELLANTRIEBIn.proModbusTest
        OnMouseClick: execute { wDetail.2 := NOT wDetail.2; }
    Label (45,70 191x20), "Bit 02 Bereitmeldung Stellantrieb"
    Textfield (5,90 20x20), "%d", text variable: TO_WORD(wDetail.3), input disabled if: NOT ITF_STELLANTRIEBIn.proModbusTest
        OnMouseClick: execute { wDetail.3 := NOT wDetail.3; }
    Label (45,90 180x20), "Bit 03 Stellanrieb ist OFFEN"
    Textfield (5,110 20x20), "%d", text variable: TO_WORD(wDetail.4), input disabled if: NOT ITF_STELLANTRIEBIn.proModbusTest
        OnMouseClick: execute { wDetail.4 := NOT wDetail.4; }
    Label (45,110 180x20), "Bit 04 Stellantrieb ist ZU"
    Textfield (5,130 20x20), "%d", text variable: TO_WORD(wDetail.5), input disabled if: NOT ITF_STELLANTRIEBIn.proModbusTest
        OnMouseClick: execute { wDetail.5 := NOT wDetail.5; }
    Label (45,130 180x20), "Bit 05 Revisionsschalter OK"
    Textfield (5,150 20x20), "%d", text variable: TO_WORD(wDetail.6), input disabled if: NOT ITF_STELLANTRIEBIn.proModbusTest
        OnMouseClick: execute { wDetail.6 := NOT wDetail.6; }
    Label (45,150 180x20), "Bit 06 Sicherung OK"
    Textfield (5,170 20x20), "%d", text variable: TO_WORD(wDetail.7), input disabled if: NOT ITF_STELLANTRIEBIn.proModbusTest
        OnMouseClick: execute { wDetail.7 := NOT wDetail.7; }
    Label (45,170 180x20), "Bit 07 Antriebsschutzschalter OK"
    Textfield (5,190 20x20), "%d", text variable: TO_WORD(wDetail.8), input disabled if: NOT ITF_STELLANTRIEBIn.proModbusTest
        OnMouseClick: execute { wDetail.8 := NOT wDetail.8; }
    Label (45,190 180x20), "Bit 08 Handmodul Aktiv"
    Textfield (5,210 20x20), "%d", text variable: TO_WORD(wDetail.9), input disabled if: NOT ITF_STELLANTRIEBIn.proModbusTest
        OnMouseClick: execute { wDetail.9 := NOT wDetail.9; }
    Label (45,210 180x20), "Bit 09 Automatikbetrieb"
    Textfield (5,230 20x20), "%d", text variable: TO_WORD(wDetail.10), input disabled if: NOT ITF_STELLANTRIEBIn.proModbusTest
        OnMouseClick: execute { wDetail.10 := NOT wDetail.10; }
    Label (45,230 180x20), "Bit 10 Reserve"
    Textfield (5,250 20x20), "%d", text variable: TO_WORD(wDetail.11), input disabled if: NOT ITF_STELLANTRIEBIn.proModbusTest
        OnMouseClick: execute { wDetail.11 := NOT wDetail.11; }
    Label (45,250 180x20), "Bit 11 Reserve"
    Textfield (5,270 20x20), "%d", text variable: TO_WORD(wDetail.12), input disabled if: NOT ITF_STELLANTRIEBIn.proModbusTest
        OnMouseClick: execute { wDetail.12 := NOT wDetail.12; }
    Label (45,270 180x20), "Bit 12 Reserve"
    Textfield (5,290 20x20), "%d", text variable: TO_WORD(wDetail.13), input disabled if: NOT ITF_STELLANTRIEBIn.proModbusTest
        OnMouseClick: execute { wDetail.13 := NOT wDetail.13; }
    Label (45,290 180x20), "Bit 13 Reserve"
    Textfield (5,310 20x20), "%d", text variable: TO_WORD(wDetail.14), input disabled if: NOT ITF_STELLANTRIEBIn.proModbusTest
        OnMouseClick: execute { wDetail.14 := NOT wDetail.14; }
    Label (45,310 180x20), "Bit 14 Warnung"
    Textfield (5,330 20x20), "%d", text variable: TO_WORD(wDetail.15), input disabled if: NOT ITF_STELLANTRIEBIn.proModbusTest
        OnMouseClick: execute { wDetail.15 := NOT wDetail.15; }
    Label (45,330 180x20), "Bit 15 Fehler"
    Image (269,0 30x30), image: LibVis01VisuBasic.imgpVisuCTA.close_solo_black
        OnMouseClick: execute { xShow := FALSE; ITF_STELLANTRIEBIN.proModbusTest := FALSE; }
    Label (5,0 150x20), "Status Word 0"
    Image (265,315 30x30), invisible if: ITF_STELLANTRIEBIN.proModbusTest, image: ImagePool.front_hand_FILL0_wght400_GRAD0_opsz48
        OnMouseClick: execute { ITF_STELLANTRIEBIN.proModbusTest := TRUE; }
    Image (265,315 30x30), invisible if: NOT ITF_STELLANTRIEBIN.proModbusTest, image: ImagePool.front_hand_FILL0_wght400_GRAD0_opsz48Yellow
        OnMouseClick: execute { ITF_STELLANTRIEBIN.proModbusTest := False; }
    Line (5,18) (265,18)
END_VISUALIZATION

// 40 Visualizations/POPUP/BUS/StellAntrieb_BUS_CW0_Detail
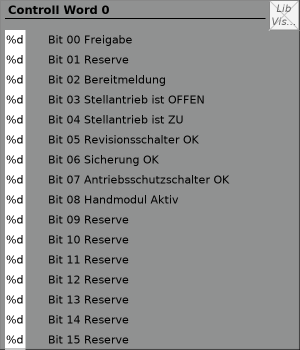
VISUALIZATION StellAntrieb_BUS_CW0_Detail  // 300x350
VAR_IN_OUT
    wDetail :   WORD;
END_VAR
VAR_IN_OUT
    xShow   :   BOOL;
END_VAR
    Rectangle (0,0 300x350)
    Textfield (5,30 20x20), "%d", text variable: TO_WORD(wDetail.0), input disabled if: TRUE
    Label (45,30 180x20), "Bit 00 Freigabe"
    Textfield (5,50 20x20), "%d", text variable: TO_WORD(wDetail.1), input disabled if: TRUE
    Label (45,50 180x20), "Bit 01 Reserve"
    Textfield (5,70 20x20), "%d", text variable: TO_WORD(wDetail.2), input disabled if: TRUE
    Label (45,70 180x20), "Bit 02 Bereitmeldung"
    Textfield (5,90 20x20), "%d", text variable: TO_WORD(wDetail.3), input disabled if: TRUE
    Label (45,90 180x20), "Bit 03 Stellantrieb ist OFFEN"
    Textfield (5,110 20x20), "%d", text variable: TO_WORD(wDetail.4), input disabled if: TRUE
    Label (45,110 180x20), "Bit 04 Stellantrieb ist ZU"
    Textfield (5,130 20x20), "%d", text variable: TO_WORD(wDetail.5), input disabled if: TRUE
    Label (45,130 180x20), "Bit 05 Revisionsschalter OK"
    Textfield (5,150 20x20), "%d", text variable: TO_WORD(wDetail.6), input disabled if: TRUE
    Label (45,150 180x20), "Bit 06 Sicherung OK"
    Textfield (5,170 20x20), "%d", text variable: TO_WORD(wDetail.7), input disabled if: TRUE
    Label (45,170 180x20), "Bit 07 Antriebsschutzschalter OK"
    Textfield (5,190 20x20), "%d", text variable: TO_WORD(wDetail.8), input disabled if: TRUE
    Label (45,190 180x20), "Bit 08 Handmodul Aktiv"
    Textfield (5,210 20x20), "%d", text variable: TO_WORD(wDetail.9), input disabled if: TRUE
    Label (45,210 180x20), "Bit 09 Reserve"
    Textfield (5,230 20x20), "%d", text variable: TO_WORD(wDetail.10), input disabled if: TRUE
    Label (45,230 180x20), "Bit 10 Reserve"
    Textfield (5,250 20x20), "%d", text variable: TO_WORD(wDetail.11), input disabled if: TRUE
    Label (45,250 180x20), "Bit 11 Reserve"
    Textfield (5,270 20x20), "%d", text variable: TO_WORD(wDetail.12), input disabled if: TRUE
    Label (45,270 180x20), "Bit 12 Reserve"
    Textfield (5,290 20x20), "%d", text variable: TO_WORD(wDetail.13), input disabled if: TRUE
    Label (45,290 180x20), "Bit 13 Reserve"
    Textfield (5,310 20x20), "%d", text variable: TO_WORD(wDetail.14), input disabled if: TRUE
    Label (45,310 180x20), "Bit 14 Reserve"
    Textfield (5,330 20x20), "%d", text variable: TO_WORD(wDetail.15), input disabled if: TRUE
    Label (45,330 180x20), "Bit 15 Reserve"
    Image (269,0 30x30), image: LibVis01VisuBasic.imgpVisuCTA.close_solo_black
        OnMouseClick: execute { xShow := FALSE; }
    Label (5,0 150x20), "Controll Word 0"
    Line (5,18) (265,18)
END_VISUALIZATION

// 40 Visualizations/POPUP/BUS/StellAntrieb_BUS_CS
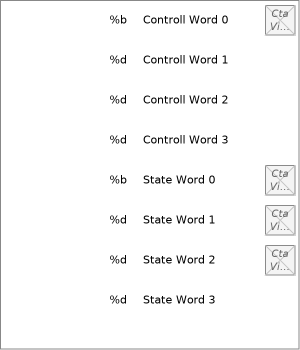
VISUALIZATION StellAntrieb_BUS_CS  // 300x350
VAR_INPUT
    ITF_STELLANTRIEBIn        :   ITF_STELLANTRIEB;
    ayControllWord  :   REFERENCE TO ARRAY[0..3] OF WORD;
    ayStateWord     :   REFERENCE TO ARRAY[0..3] OF WORD;
END_VAR
VAR
    xShowCw :   BOOL;
    xShowSw :   BOOL;
    xShowSw1:   BOOL;
    xShowSw2:   BOOL;
END_VAR
    Textfield (0,10 130x20), "%b", text variable: ayControllWord[0]
    Label (140,10 120x20), "Controll Word 0"
    Label (140,50 120x20), "Controll Word 1"
    Textfield (0,50 130x20), "%d", text variable: ayControllWord[1]
    Label (140,90 120x20), "Controll Word 2", invisible if: TRUE
    Textfield (0,90 130x20), "%d", text variable: ayControllWord[2], invisible if: TRUE
    Label (140,130 120x20), "Controll Word 3", invisible if: TRUE
    Textfield (0,130 130x20), "%d", text variable: ayControllWord[2], invisible if: TRUE
    Image (265,5 30x30), image: CtaVisSymbols.ImagePool.information-variant
        OnMouseClick: execute {
            xShowCw := TRUE;
            xShowSw := FALSE;
            xShowSw1:= FALSE;
            xShowSw2:= FALSE;
        }
    Frame (300,0 300x350), invisible if: NOT xShowCw
        shows StellAntrieb_BUS_CW0_Detail(wDetail := ayControllWord[0], xShow := xShowCw)
    Label (140,290 120x20), "State Word 3", invisible if: TRUE
    Textfield (0,170 130x20), "%b", text variable: ayStateWord[0]
        OnMouseDown: write the text variable via Default
    Label (140,170 120x20), "State Word 0"
    Label (140,210 120x20), "State Word 1"
    Textfield (0,210 130x20), "%d", text variable: ayStateWord[1]
    Label (140,250 120x20), "State Word 2"
    Textfield (0,250 130x20), "%d", text variable: ayStateWord[2]
    Textfield (0,290 130x20), "%d", text variable: ayStateWord[2], invisible if: TRUE
    Image (265,165 30x30), image: CtaVisSymbols.ImagePool.information-variant
        OnMouseClick: execute {
            xShowCw := FALSE;
            xShowSw := TRUE;
            xShowSw1:= FALSE;
            xShowSw2:= FALSE;
        }
    Frame (300,0 300x350), invisible if: NOT xShowSw
        shows StellAntrieb_BUS_SW0_Detail(wDetail := ayStateWord[0], ITF_STELLANTRIEBIN := ITF_STELLANTRIEBIN, xShow := xShowSw2)
    Image (265,205 30x30), image: CtaVisSymbols.ImagePool.information-variant
        OnMouseClick: execute {
            xShowCw := FALSE;
            xShowSw := FALSE;
            xShowSw1:= TRUE;
            xShowSw2:= FALSE;
        }
    Frame (300,0 300x350), invisible if: NOT xShowSw1
        shows StellAntrieb_BUS_SW1_Detail(wDetail := ayStateWord[1], ITF_STELLANTRIEBIN := ITF_STELLANTRIEBIn, xShow := xShowSw1)
    Frame (300,0 300x350), invisible if: NOT xShowSw2
        shows StellAntrieb_BUS_SW2_Detail(wDetail := ayStateWord[2], ITF_STELLANTRIEBIN := ITF_STELLANTRIEBIn, xShow := xShowSw2)
    Image (265,245 30x30), image: CtaVisSymbols.ImagePool.information-variant
        OnMouseClick: execute {
            xShowCw := FALSE;
            xShowSw := FALSE;
            xShowSw1:= FALSE;
            xShowSw2:= TRUE;
        }
END_VISUALIZATION

// 40 Visualizations/POPUP/BUS/StellAntrieb_BUS_SW1_Detail
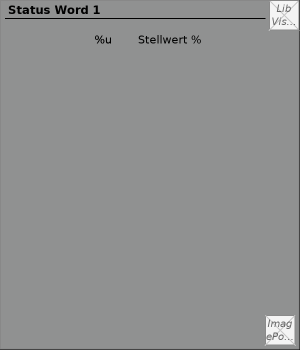
VISUALIZATION StellAntrieb_BUS_SW1_Detail  // 300x350
VAR_IN_OUT
    wDetail     :   WORD;
END_VAR
VAR_INPUT	
    ITF_STELLANTRIEBIN    :   ITF_STELLANTRIEB;
END_VAR
VAR_IN_OUT
    xShow       :   BOOL;
END_VAR
    Rectangle (0,0 300x350)
    Image (269,0 30x30), image: LibVis01VisuBasic.imgpVisuCTA.close_solo_black
        OnMouseClick: execute { xShow := FALSE; ITF_STELLANTRIEBIN.proModbusTest := FALSE; }
    Label (5,0 150x20), "Status Word 1"
    Image (265,315 30x30), invisible if: ITF_STELLANTRIEBIN.proModbusTest, image: ImagePool.front_hand_FILL0_wght400_GRAD0_opsz48
        OnMouseClick: execute { ITF_STELLANTRIEBIN.proModbusTest := TRUE; }
    Image (265,315 30x30), invisible if: NOT ITF_STELLANTRIEBIn.proModbusTest, image: ImagePool.front_hand_FILL0_wght400_GRAD0_opsz48Yellow
        OnMouseClick: execute { ITF_STELLANTRIEBIN.proModbusTest := False; }
    Label (135,30 120x20), "Stellwert %"
    Textfield (5,30 110x20), "%u", text variable: wDetail, input disabled if: NOT ITF_STELLANTRIEBIn.proModbusTest
        OnMouseClick: write the text variable via InputWithLimits, min 0, max 100
    Textfield (5,30 110x20), "%u", text variable: wDetail, invisible if: ITF_STELLANTRIEBIN.proModbusTest
    Line (5,18) (265,18)
END_VISUALIZATION

// 40 Visualizations/POPUP/BUS/StellAntrieb_BUS_SW2_Detail
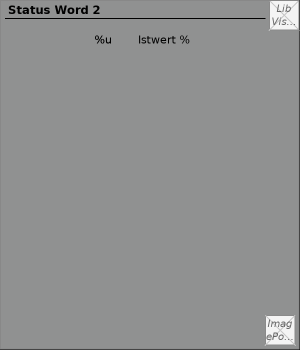
VISUALIZATION StellAntrieb_BUS_SW2_Detail  // 300x350
VAR_IN_OUT
    wDetail             :   WORD;
END_VAR
VAR_INPUT	
    ITF_STELLANTRIEBIN       :   ITF_STELLANTRIEB;
END_VAR
VAR_IN_OUT
    xShow               :   BOOL;
END_VAR
    Rectangle (0,0 300x350)
    Image (269,0 30x30), image: LibVis01VisuBasic.imgpVisuCTA.close_solo_black
        OnMouseClick: execute { xShow := FALSE; ITF_STELLANTRIEBIN.proModbusTest := FALSE; }
    Label (5,0 150x20), "Status Word 2"
    Image (265,315 30x30), invisible if: ITF_STELLANTRIEBIn.proModbusTest, image: ImagePool.front_hand_FILL0_wght400_GRAD0_opsz48
        OnMouseClick: execute { ITF_STELLANTRIEBIN.proModbusTest := TRUE; }
    Image (265,315 30x30), invisible if: NOT ITF_STELLANTRIEBIN.proModbusTest, image: ImagePool.front_hand_FILL0_wght400_GRAD0_opsz48Yellow
        OnMouseClick: execute { ITF_STELLANTRIEBIN.proModbusTest := False; }
    Label (135,30 120x20), "Istwert %"
    Textfield (5,30 110x20), "%u", text variable: wDetail, input disabled if: NOT ITF_STELLANTRIEBIn.proModbusTest
        OnMouseClick: write the text variable via InputWithLimits, min 0, max 100
    Textfield (5,30 110x20), "%u", text variable: wDetail, invisible if: ITF_STELLANTRIEBIN.proModbusTest
    Line (5,18) (265,18)
END_VISUALIZATION

// 40 Visualizations/POPUP/REPORTS/StellAntrieb_REPORTS
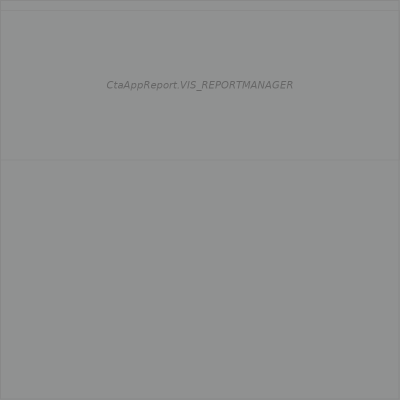
VISUALIZATION StellAntrieb_REPORTS  // 400x400
VAR_INPUT
    ITF_STELLANTRIEBIN    :   ITF_STELLANTRIEB;	
END_VAR
    Frame (0,10 400x150)
        shows CtaAppReport.VIS_REPORTMANAGER(ITF_REPORTMANAGER := ITF_STELLANTRIEBIN.proITF_REPORTMANAGER)
END_VISUALIZATION

// 40 Visualizations/POPUP/PARAMETER/StellAntrieb_ParameterBase/StellAntrieb_ParameterBase0
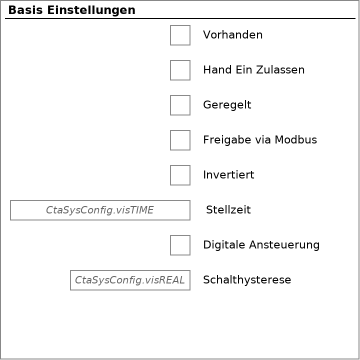
VISUALIZATION StellAntrieb_ParameterBase0  // 360x360
VAR_INPUT
    ITF_STELLANTRIEBIN : ITF_STELLANTRIEB;
END_VAR
    Label (5,0 350x20), "Basis Einstellungen"
    Frame (170,25 20x20)
        shows CtaSysConfig.visBOOL(visfbBOOLIn := ITF_STELLANTRIEBIN.p_scBase_fbxEnable)
    Label (200,25 150x20), "Vorhanden"
    Frame (170,95 20x20)
        shows CtaSysConfig.visBOOL(visfbBOOLIn := ITF_STELLANTRIEBIN.p_scBase_fbxRegulatet)
    Label (200,95 150x20), "Geregelt"
    Label (200,130 150x20), "Freigabe via Modbus"
    Frame (170,130 20x20)
        shows CtaSysConfig.visBOOL(visfbBOOLIn := ITF_STELLANTRIEBIN.p_scBase_fbxControllMb)
    Frame (170,60 20x20)
        shows CtaSysConfig.visBOOL(visfbBOOLIn := ITF_STELLANTRIEBIN.p_scManual_fbxAlowManualOn)
    Label (200,60 150x20), "Hand Ein Zulassen"
    Frame (170,165 20x20)
        shows CtaSysConfig.visBOOL(visfbBOOLIn := ITF_STELLANTRIEBIN.p_scBase_fbxInvertiert)
    Label (200,165 150x20), "Invertiert"
    Frame (10,200 180x20)
        shows CtaSysConfig.visTIME(visfbTIMEIn := ITF_STELLANTRIEBIN.p_scBase_fbtYSettingTime)
    Label (203,200 150x20), "Stellzeit"
    Label (200,235 150x20), "Digitale Ansteuerung"
    Frame (70,270 120x20)
        shows CtaSysConfig.visREAL(visfbREALIn := ITF_STELLANTRIEBIN.p_scBase_fbrHysteresisDigital, stPhysikalischeEinheit := '%')
    Label (200,270 150x20), "Schalthysterese"
    Frame (170,235 20x20)
        shows CtaSysConfig.visBOOL(visfbBOOLIn := ITF_STELLANTRIEBIN.p_scBase_fbxEnDigitalValve)
    Line (5,18) (355,18)
END_VISUALIZATION

// 40 Visualizations/POPUP/PARAMETER/StellAntrieb_ParameterBase/StellAntrieb_ParameterBase
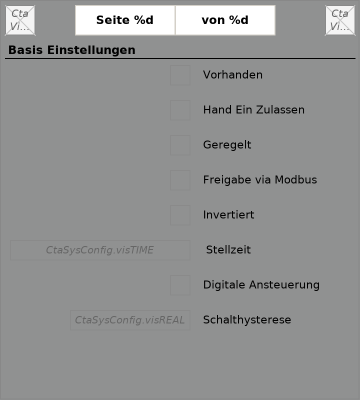
VISUALIZATION StellAntrieb_ParameterBase  // 360x400
VAR_INPUT
    ITF_STELLANTRIEBIN : ITF_STELLANTRIEB;
END_VAR
VAR
    uiPage  :   UINT;
    uiMin   :   UINT    := 0;
    uiMax   :   UINT    := 2;
END_VAR
    Image (5,5 30x30), invisible if: uiPage = uiMin, image: CtaVisSymbols.ImagePool.arrow-left_square
        OnMouseClick: execute {
            uiPage := uiPage - 1;
            IF uiPage <= uiMin THEN
                uiPage := uiMin;
            END_IF;
        }
    Image (325,5 30x30), invisible if: uiPage = uiMax, image: CtaVisSymbols.ImagePool.arrow-right_square
        OnMouseClick: execute {
            uiPage := uiPage + 1;
            IF uiPage >= uiMax THEN
                uiPage := uiMax;
            END_IF;
        }
    Frame (0,40 360x360), frame switch variable: uiPage
        shows StellAntrieb_ParameterBase0(ITF_STELLANTRIEBIN := ITF_STELLANTRIEBIN)
        shows StellAntrieb_ParameterBase1(ITF_STELLANTRIEBIN := ITF_STELLANTRIEBIN)
        shows StellAntrieb_ParameterBase2(ITF_STELLANTRIEBIN := ITF_STELLANTRIEBIN)
        shows StellAntrieb_ParameterBase2()
        pReferences[0]: ITF_Parameter=ITF_Parameter
        p2498127594: ITF_Parameter
    Textfield (175,5 100x30), "von %d", text variable: uiMax
    Textfield (75,5 100x30), "Seite %d", text variable: uiPage
END_VISUALIZATION

// 40 Visualizations/POPUP/PARAMETER/StellAntrieb_Fuse/StellAntrieb_ParameterFuses0
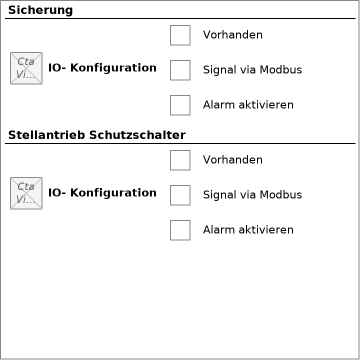
VISUALIZATION StellAntrieb_ParameterFuses0  // 360x360
VAR_INPUT
    ITF_STELLANTRIEBIN 	:	ITF_STELLANTRIEB;
	ITF_Fuse_IN 		:	CtaSysIO.ITF_IO;
	ITF_ActuatorFuse_IN 	:	CtaSysIO.ITF_IO;
END_VAR
    Frame (170,25 20x20)
        shows CtaSysConfig.visBOOL(visfbBOOLIn := ITF_STELLANTRIEBIN.p_scFuse_fbxEnable)
    Label (200,25 150x20), "Vorhanden"
    Frame (170,60 20x20)
        shows CtaSysConfig.visBOOL(visfbBOOLIn := ITF_STELLANTRIEBIN.p_scFuse_fbxInputMb)
    Label (200,60 150x20), "Signal via Modbus"
    Frame (170,95 20x20)
        shows CtaSysConfig.visBOOL(visfbBOOLIn := ITF_STELLANTRIEBIN.p_scFuse_fbxDoesAlarm)
    Label (200,95 150x20), "Alarm aktivieren"
    Label (5,0 350x20), "Sicherung"
    Label (5,125 350x20), "Stellantrieb Schutzschalter"
    Frame (170,150 20x20)
        shows CtaSysConfig.visBOOL(visfbBOOLIn := ITF_STELLANTRIEBIN.p_scActuatorFuse_fbxEnable)
    Label (200,150 150x20), "Vorhanden"
    Frame (170,185 20x20)
        shows CtaSysConfig.visBOOL(visfbBOOLIn := ITF_STELLANTRIEBIN.p_scActuatorFuse_fbxInputMb)
    Label (200,185 150x20), "Signal via Modbus"
    Frame (170,220 20x20)
        shows CtaSysConfig.visBOOL(visfbBOOLIn := ITF_STELLANTRIEBIN.p_scActuatorFuse_fbxDoesAlarm)
    Label (200,220 150x20), "Alarm aktivieren"
    Line (5,18) (355,18)
    Line (5,143) (355,143)
    Label (45,58 120x20), "IO- Konfiguration", invisible if: ITF_Fuse_IN = 0
    Image (10,52 32x32), invisible if: ITF_Fuse_IN = 0, image: CtaVisSymbols.ImagePool.build
        OnMouseDown:  Dialog=StellAntrieb_POPUP_IO_ITF, Parameters={ITF_IO_IN: ITF_Fuse_IN}, OpenModal=True, OpenCentered=True
    Image (10,177 32x32), invisible if: ITF_ActuatorFuse_IN = 0, image: CtaVisSymbols.ImagePool.build
        OnMouseDown:  Dialog=StellAntrieb_POPUP_IO_ITF, Parameters={ITF_IO_IN: ITF_ActuatorFuse_IN}, OpenModal=True, OpenCentered=True
    Label (45,183 120x20), "IO- Konfiguration", invisible if: ITF_ActuatorFuse_IN = 0
END_VISUALIZATION

// 40 Visualizations/POPUP/PARAMETER/StellAntrieb_Fuse/StellAntrieb_ParameterFuses
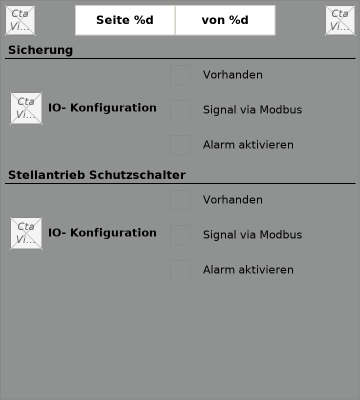
VISUALIZATION StellAntrieb_ParameterFuses  // 360x400
VAR_INPUT
    ITF_STELLANTRIEBIN : ITF_STELLANTRIEB;
END_VAR
VAR
    uiPage  :   UINT;
    uiMin   :   UINT    := 0;
    uiMax   :   UINT    := 0;
END_VAR
    Image (5,5 30x30), invisible if: uiPage = uiMin, image: CtaVisSymbols.ImagePool.arrow-left_square
        OnMouseClick: execute {
            uiPage := uiPage - 1;
            IF uiPage <= uiMin THEN
                uiPage := uiMin;
            END_IF;
        }
    Image (325,5 30x30), invisible if: uiPage = uiMax, image: CtaVisSymbols.ImagePool.arrow-right_square
        OnMouseClick: execute {
            uiPage := uiPage + 1;
            IF uiPage >= uiMax THEN
                uiPage := uiMax;
            END_IF;
        }
    Frame (0,40 360x360), frame switch variable: uiPage
        shows StellAntrieb_ParameterFuses0(ITF_STELLANTRIEBIN := ITF_STELLANTRIEBIN, ITF_Fuse_IN := ITF_STELLANTRIEBIN.proFuse_ITF, ITF_ActuatorFuse_IN := ITF_STELLANTRIEBIN.proActuatorFuse_ITF)
        shows AT_ParameterIO1(ITF_Parameter := ITF_Parameter)
        pReferences[0]: ITF_Parameter=ITF_Parameter
    Textfield (75,5 100x30), "Seite %d", text variable: uiPage
    Textfield (175,5 100x30), "von %d", text variable: uiMax
END_VISUALIZATION

// 40 Visualizations/POPUP/PARAMETER/StellAntrieb_IO/StellAntrieb_ParameterIO0
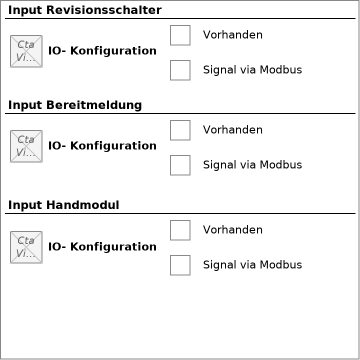
VISUALIZATION StellAntrieb_ParameterIO0  // 360x360
VAR_INPUT
    ITF_STELLANTRIEBIN 	:	ITF_STELLANTRIEB;
	ITF_RevSwitch_IN 	:	CtaSysIO.ITF_IO;
	ITF_Ready_IN		:	CtaSysIO.ITF_IO;
	ITF_HandModul_IN 	:	CtaSysIO.ITF_IO;
END_VAR
    Frame (170,25 20x20)
        shows CtaSysConfig.visBOOL(visfbBOOLIn := ITF_STELLANTRIEBIN.p_scInStellAtRevisionSwitch_fbxEnable)
    Label (200,25 150x20), "Vorhanden"
    Frame (170,60 20x20)
        shows CtaSysConfig.visBOOL(visfbBOOLIn := ITF_STELLANTRIEBIN.p_scInStellAtRevisionSwitch_fbxInputMb)
    Label (200,60 150x20), "Signal via Modbus"
    Label (5,0 350x20), "Input Revisionsschalter"
    Label (5,95 350x20), "Input Bereitmeldung"
    Frame (170,120 20x20)
        shows CtaSysConfig.visBOOL(visfbBOOLIn := ITF_STELLANTRIEBIN.p_scInStellAtReady_fbxEnable)
    Label (200,120 150x20), "Vorhanden"
    Frame (170,155 20x20)
        shows CtaSysConfig.visBOOL(visfbBOOLIn := ITF_STELLANTRIEBIN.p_scInStellAtReady_fbxInputMb)
    Label (200,155 150x20), "Signal via Modbus"
    Label (5,195 350x20), "Input Handmodul"
    Frame (170,220 20x20)
        shows CtaSysConfig.visBOOL(visfbBOOLIn := ITF_STELLANTRIEBIN.p_scInStellAtHand_fbxEnable)
    Label (200,220 150x20), "Vorhanden"
    Frame (170,255 20x20)
        shows CtaSysConfig.visBOOL(visfbBOOLIn := ITF_STELLANTRIEBIN.p_scInStellAtHand_fbxInputMb)
    Label (200,255 150x20), "Signal via Modbus"
    Line (5,18) (355,18)
    Line (5,113) (355,113)
    Line (5,213) (355,213)
    Image (10,35 32x32), invisible if: ITF_RevSwitch_IN = 0, image: CtaVisSymbols.ImagePool.build
        OnMouseDown:  Dialog=StellAntrieb_POPUP_IO_ITF, Parameters={ITF_IO_IN: ITF_RevSwitch_IN}, OpenModal=True, OpenCentered=True
    Label (45,41 120x20), "IO- Konfiguration", invisible if: ITF_RevSwitch_IN = 0
    Image (10,130 32x32), invisible if: ITF_Ready_IN = 0, image: CtaVisSymbols.ImagePool.build
        OnMouseDown:  Dialog=StellAntrieb_POPUP_IO_ITF, Parameters={ITF_IO_IN: ITF_Ready_IN}, OpenModal=True, OpenCentered=True
    Label (45,136 120x20), "IO- Konfiguration", invisible if: ITF_Ready_IN = 0
    Image (10,231 32x32), invisible if: ITF_HandModul_IN = 0, image: CtaVisSymbols.ImagePool.build
        OnMouseDown:  Dialog=StellAntrieb_POPUP_IO_ITF, Parameters={ITF_IO_IN: ITF_HandModul_IN}, OpenModal=True, OpenCentered=True
    Label (45,237 120x20), "IO- Konfiguration", invisible if: ITF_HandModul_IN = 0
END_VISUALIZATION

// 40 Visualizations/POPUP/PARAMETER/StellAntrieb_IO/StellAntrieb_ParameterIO1
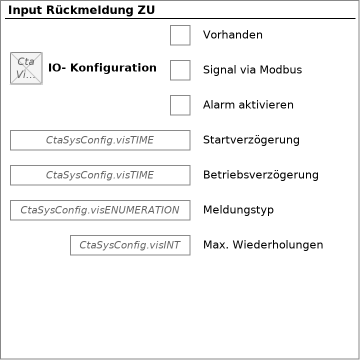
VISUALIZATION StellAntrieb_ParameterIO1  // 360x360
VAR_INPUT
    ITF_STELLANTRIEBIN 	:	ITF_STELLANTRIEB;
	ITF_RückClosed_IN	:	CtaSysIO.ITF_IO;
END_VAR
    Label (5,0 350x20), "Input Rückmeldung ZU"
    Frame (170,25 20x20)
        shows CtaSysConfig.visBOOL(visfbBOOLIn := ITF_STELLANTRIEBIN.p_scInStellAtRükClosed_fbxEnable)
    Label (200,25 150x20), "Vorhanden"
    Frame (170,60 20x20)
        shows CtaSysConfig.visBOOL(visfbBOOLIn := ITF_STELLANTRIEBIN.p_scInStellAtRükClosed_fbxInputMb)
    Label (200,60 150x20), "Signal via Modbus"
    Frame (170,95 20x20)
        shows CtaSysConfig.visBOOL(visfbBOOLIn := ITF_STELLANTRIEBIN.p_scInStellAtRükClosed_fbxDoesAlarm)
    Label (200,95 150x20), "Alarm aktivieren"
    Frame (10,130 180x20)
        shows CtaSysConfig.visTIME(visfbTIMEIn := ITF_STELLANTRIEBIN.p_scInStellAtRükClosed_fbtDelayStart)
    Label (200,130 150x20), "Startverzögerung"
    Label (200,165 150x20), "Betriebsverzögerung"
    Frame (10,165 180x20)
        shows CtaSysConfig.visTIME(visfbTIMEIn := ITF_STELLANTRIEBIN.p_scInStellAtRükClosed_fbtDelayRun)
    Label (200,200 150x20), "Meldungstyp"
    Label (200,235 150x20), "Max. Wiederholungen"
    Line (5,18) (355,18)
    Frame (10,200 180x20), text list: 'CtaAppReport.txtLibAp99_2enTypeOfAck', text index: CtaSysConfig.fcGetEnumerationId(ITF_STELLANTRIEBIN.p_scInStellAtRükClosed_fbiTypeOfAck)
        shows CtaSysConfig.visENUMERATION(visfbENUIn := ITF_STELLANTRIEBIN.p_scInStellAtRükClosed_fbiTypeOfAck)
    Frame (70,235 120x20)
        shows CtaSysConfig.visINT(visfbINTIn := ITF_STELLANTRIEBIN.p_scInStellAtRükClosed_fbiMaxErrorRetryAllowed)
    Image (10,52 32x32), invisible if: ITF_RückClosed_IN = 0, image: CtaVisSymbols.ImagePool.build
        OnMouseDown:  Dialog=StellAntrieb_POPUP_IO_ITF, Parameters={ITF_IO_IN: ITF_RückClosed_IN}, OpenModal=True, OpenCentered=True
    Label (45,58 120x20), "IO- Konfiguration", invisible if: ITF_RückClosed_IN = 0
END_VISUALIZATION

// 40 Visualizations/POPUP/PARAMETER/StellAntrieb_IO/StellAntrieb_ParameterIO
